LIN {X 0,Y 298.545,Z 280.112,A -85,B 0,C 180,E1 -16213.618,E2 -16213.618} C_VEL
LIN {X 0,Y 298.541,Z 280.111,A -85,B 0,C 180,E1 -16216.411,E2 -16216.411} C_VEL
LIN {X 0,Y 298.503,Z 280.117,A -85,B 0,C 180,E1 -16219.656,E2 -16219.656} C_VEL
LIN {X 0,Y 298.417,Z 280.126,A -85,B 0,C 180,E1 -16223.603,E2 -16223.603} C_VEL
LIN {X 0,Y 298.403,Z 280.131,A -85,B 0,C 180,E1 -16226.585,E2 -16226.585} C_VEL
LIN {X 0,Y 298.388,Z 280.134,A -85,B 0,C 180,E1 -16229.647,E2 -16229.647} C_VEL
LIN {X 0,Y 298.388,Z 280.135,A -85,B 0,C 180,E1 -16232.803,E2 -16232.803} C_VEL
LIN {X 0,Y 298.461,Z 280.124,A -85,B 0,C 180,E1 -16236.815,E2 -16236.815} C_VEL
LIN {X 0,Y 298.415,Z 280.127,A -85,B 0,C 180,E1 -16241.097,E2 -16241.097} C_VEL
LIN {X 0,Y 298.427,Z 280.25,A -85,B 0,C 180,E1 -16243.54,E2 -16243.54} C_VEL
LIN {X 0,Y 299.046,Z 283.99,A -85,B 0,C 180,E1 -16247.039,E2 -16247.039} C_VEL
LIN {X 0,Y 299.67,Z 287.19,A -85,B 0,C 180,E1 -16249.842,E2 -16249.842} C_VEL
LIN {X 0,Y 300.261,Z 290.689,A -85,B 0,C 180,E1 -16252.735,E2 -16252.735} C_VEL
LIN {X 0,Y 300.627,Z 293.494,A -85,B 0,C 180,E1 -16254.91,E2 -16254.91} C_VEL
LIN {X 0,Y 300.519,Z 296.811,A -85,B 0,C 180,E1 -16257.344,E2 -16257.344} C_VEL
LIN {X 0,Y 299.5,Z 302.518,A -85,B 0,C 180,E1 -16261.248,E2 -16261.248} C_VEL
LIN {X 0,Y 298.415,Z 309.186,A -85,B 0,C 180,E1 -16265.663,E2 -16265.663} C_VEL
LIN {X 0,Y 297.791,Z 313.823,A -85,B 0,C 180,E1 -16268.636,E2 -16268.636} C_VEL
LIN {X 0,Y 300.523,Z 326.073,A -85,B 0,C 180,E1 -16269.564,E2 -16269.564} C_VEL
LIN {X 0,Y 302.121,Z 336.168,A -85,B 0,C 180,E1 -16270.52,E2 -16270.52} C_VEL
LIN {X 0,Y 302.918,Z 345.087,A -85,B 0,C 180,E1 -16271.519,E2 -16271.519} C_VEL
LIN {X 0,Y 303.106,Z 352.307,A -85,B 0,C 180,E1 -16272.459,E2 -16272.459} C_VEL
LIN {X 0,Y 302.625,Z 359.174,A -85,B 0,C 180,E1 -16273.474,E2 -16273.474} C_VEL
LIN {X 0,Y 301.244,Z 366.76,A -85,B 0,C 180,E1 -16274.786,E2 -16274.786} C_VEL
LIN {X 0,Y 300.07,Z 373.019,A -85,B 0,C 180,E1 -16276.111,E2 -16276.111} C_VEL
LIN {X 0,Y 299.132,Z 378.235,A -85,B 0,C 180,E1 -16277.45,E2 -16277.45} C_VEL
LIN {X 0,Y 298.133,Z 383.56,A -85,B 0,C 180,E1 -16279.132,E2 -16279.132} C_VEL
LIN {X 0,Y 297.531,Z 387.015,A -85,B 0,C 180,E1 -16280.484,E2 -16280.484} C_VEL
LIN {X 0,Y 296.906,Z 391.022,A -85,B 0,C 180,E1 -16282.521,E2 -16282.521} C_VEL
LIN {X 0,Y 296.605,Z 393.796,A -85,B 0,C 180,E1 -16284.563,E2 -16284.563} C_VEL
LIN {X 0,Y 296.606,Z 394.925,A -85,B 0,C 180,E1 -16285.926,E2 -16285.926} C_VEL
LIN {X 0,Y 296.591,Z 395.588,A -85,B 0,C 180,E1 -16287.285,E2 -16287.285} C_VEL
LIN {X 0,Y 296.599,Z 395.794,A -85,B 0,C 180,E1 -16288.644,E2 -16288.644} C_VEL
LIN {X 0,Y 296.676,Z 395.491,A -85,B 0,C 180,E1 -16290.002,E2 -16290.002} C_VEL
LIN {X 0,Y 296.641,Z 394.591,A -85,B 0,C 180,E1 -16291.359,E2 -16291.359} C_VEL
LIN {X 0,Y 296.633,Z 393.199,A -85,B 0,C 180,E1 -16292.718,E2 -16292.718} C_VEL
LIN {X 0,Y 296.668,Z 390.135,A -85,B 0,C 180,E1 -16294.758,E2 -16294.758} C_VEL
LIN {X 0,Y 296.805,Z 385.735,A -85,B 0,C 180,E1 -16296.801,E2 -16296.801} C_VEL
LIN {X 0,Y 297.112,Z 380.807,A -85,B 0,C 180,E1 -16298.503,E2 -16298.503} C_VEL
LIN {X 0,Y 297.524,Z 374.552,A -85,B 0,C 180,E1 -16300.206,E2 -16300.206} C_VEL
LIN {X 0,Y 298.089,Z 368.449,A -85,B 0,C 180,E1 -16301.562,E2 -16301.562} C_VEL
LIN {X 0,Y 298.72,Z 362.048,A -85,B 0,C 180,E1 -16302.744,E2 -16302.744} C_VEL
LIN {X 0,Y 299.405,Z 354.282,A -85,B 0,C 180,E1 -16303.924,E2 -16303.924} C_VEL
LIN {X 0,Y 299.61,Z 349.093,A -85,B 0,C 180,E1 -16304.607,E2 -16304.607} C_VEL
LIN {X 0,Y 299.163,Z 340.12,A -85,B 0,C 180,E1 -16305.592,E2 -16305.592} C_VEL
LIN {X 0,Y 298.532,Z 330.671,A -85,B 0,C 180,E1 -16306.411,E2 -16306.411} C_VEL
LIN {X 0,Y 297.725,Z 321.328,A -85,B 0,C 180,E1 -16307.031,E2 -16307.031} C_VEL
LIN {X 0,Y 296.991,Z 314.602,A -85,B 0,C 180,E1 -16307.385,E2 -16307.385} C_VEL
LIN {X 0,Y 297.477,Z 307.895,A -85,B 0,C 180,E1 -16311.483,E2 -16311.483} C_VEL
LIN {X 0,Y 298.201,Z 300.922,A -85,B 0,C 180,E1 -16315.785,E2 -16315.785} C_VEL
LIN {X 0,Y 299.154,Z 293.722,A -85,B 0,C 180,E1 -16320.34,E2 -16320.34} C_VEL
LIN {X 0,Y 299.771,Z 290.127,A -85,B 0,C 180,E1 -16322.633,E2 -16322.633} C_VEL
LIN {X 0,Y 299.704,Z 286.87,A -85,B 0,C 180,E1 -16324.838,E2 -16324.838} C_VEL
LIN {X 0,Y 298.969,Z 282.858,A -85,B 0,C 180,E1 -16327.678,E2 -16327.678} C_VEL
LIN {X 0,Y 298.502,Z 280.116,A -85,B 0,C 180,E1 -16329.692,E2 -16329.692} C_VEL
LIN {X 0,Y 298.41,Z 280.124,A -85,B 0,C 180,E1 -16333.103,E2 -16333.103} C_VEL
LIN {X 0,Y 298.414,Z 280.123,A -85,B 0,C 180,E1 -16336.921,E2 -16336.921} C_VEL
LIN {X 0,Y 298.415,Z 280.123,A -85,B 0,C 180,E1 -16341.006,E2 -16341.006} C_VEL
LIN {X 0,Y 298.429,Z 280.124,A -85,B 0,C 180,E1 -16343.93,E2 -16343.93} C_VEL
LIN {X 0,Y 298.406,Z 280.125,A -85,B 0,C 180,E1 -16347.983,E2 -16347.983} C_VEL
LIN {X 0,Y 298.474,Z 280.117,A -85,B 0,C 180,E1 -16351.903,E2 -16351.903} C_VEL
LIN {X 0,Y 298.494,Z 280.115,A -85,B 0,C 180,E1 -16354.923,E2 -16354.923} C_VEL
LIN {X 0,Y 298.433,Z 280.125,A -85,B 0,C 180,E1 -16359.312,E2 -16359.312} C_VEL
LIN {X 0,Y 298.476,Z 280.115,A -85,B 0,C 180,E1 -16362.173,E2 -16362.173} C_VEL
LIN {X 0,Y 298.595,Z 280.105,A -85,B 0,C 180,E1 -16364.993,E2 -16364.993} C_VEL
LIN {X 0,Y 298.592,Z 280.103,A -85,B 0,C 180,E1 -16369.144,E2 -16369.144} C_VEL
LIN {X 0,Y 298.726,Z 280.084,A -85,B 0,C 180,E1 -16371.883,E2 -16371.883} C_VEL
LIN {X 0,Y 298.66,Z 280.096,A -85,B 0,C 180,E1 -16374.597,E2 -16374.597} C_VEL
LIN {X 0,Y 298.929,Z 280.062,A -85,B 0,C 180,E1 -16378.65,E2 -16378.65} C_VEL
LIN {X 0,Y 298.93,Z 280.058,A -85,B 0,C 180,E1 -16381.345,E2 -16381.345} C_VEL
LIN {X 0,Y 298.803,Z 280.076,A -85,B 0,C 180,E1 -16386.751,E2 -16386.751} C_VEL
LIN {X 0,Y 298.685,Z 280.088,A -85,B 0,C 180,E1 -16389.478,E2 -16389.478} C_VEL
LIN {X 0,Y 298.555,Z 280.106,A -85,B 0,C 180,E1 -16393.612,E2 -16393.612} C_VEL
LIN {X 0,Y 298.551,Z 280.109,A -85,B 0,C 180,E1 -16396.406,E2 -16396.406} C_VEL
LIN {X 0,Y 298.513,Z 280.112,A -85,B 0,C 180,E1 -16399.651,E2 -16399.651} C_VEL
LIN {X 0,Y 298.458,Z 280.119,A -85,B 0,C 180,E1 -16403.594,E2 -16403.594} C_VEL
LIN {X 0,Y 298.486,Z 280.114,A -85,B 0,C 180,E1 -16406.571,E2 -16406.571} C_VEL
LIN {X 0,Y 298.414,Z 280.127,A -85,B 0,C 180,E1 -16409.638,E2 -16409.638} C_VEL
LIN {X 0,Y 298.392,Z 280.126,A -85,B 0,C 180,E1 -16412.797,E2 -16412.797} C_VEL
LIN {X 0,Y 298.467,Z 280.117,A -85,B 0,C 180,E1 -16416.81,E2 -16416.81} C_VEL
LIN {X 0,Y 298.451,Z 280.122,A -85,B 0,C 180,E1 -16421.246,E2 -16421.246} C_VEL
LIN {X 0,Y 298.483,Z 280.118,A -85,B 0,C 180,E1 -16425.057,E2 -16425.057} C_VEL
LIN {X 0,Y 298.445,Z 280.122,A -85,B 0,C 180,E1 -16428.895,E2 -16428.895} C_VEL
LIN {X 0,Y 298.456,Z 280.121,A -85,B 0,C 180,E1 -16433.184,E2 -16433.184} C_VEL
LIN {X 0,Y 298.385,Z 280.129,A -85,B 0,C 180,E1 -16437.197,E2 -16437.197} C_VEL
LIN {X 0,Y 298.42,Z 280.126,A -85,B 0,C 180,E1 -16440.612,E2 -16440.612} C_VEL
LIN {X 0,Y 298.472,Z 280.116,A -85,B 0,C 180,E1 -16443.471,E2 -16443.471} C_VEL
LIN {X 0,Y 298.425,Z 280.126,A -85,B 0,C 180,E1 -16446.693,E2 -16446.693} C_VEL
LIN {X 0,Y 298.418,Z 280.125,A -85,B 0,C 180,E1 -16450.747,E2 -16450.747} C_VEL
LIN {X 0,Y 298.015,Z 280.174,A -85,B 0,C 180,E1 -16454.963,E2 -16454.963} C_VEL
LIN {X 0,Y 297.655,Z 280.391,A -85,B 0,C 180,E1 -16457.383,E2 -16457.383} C_VEL
LIN {X 0,Y 297.631,Z 285.417,A -85,B 0,C 180,E1 -16462.607,E2 -16462.607} C_VEL
LIN {X 0,Y 297.388,Z 289.552,A -85,B 0,C 180,E1 -16466.781,E2 -16466.781} C_VEL
LIN {X 0,Y 299.242,Z 300.537,A -85,B 0,C 180,E1 -16467.474,E2 -16467.474} C_VEL
LIN {X 0,Y 300.308,Z 308.84,A -85,B 0,C 180,E1 -16468.154,E2 -16468.154} C_VEL
LIN {X 0,Y 301.049,Z 315.665,A -85,B 0,C 180,E1 -16468.828,E2 -16468.828} C_VEL
LIN {X 0,Y 300.195,Z 325.606,A -85,B 0,C 180,E1 -16469.998,E2 -16469.998} C_VEL
LIN {X 0,Y 299.521,Z 333.548,A -85,B 0,C 180,E1 -16471.175,E2 -16471.175} C_VEL
LIN {X 0,Y 298.889,Z 340.115,A -85,B 0,C 180,E1 -16472.357,E2 -16472.357} C_VEL
LIN {X 0,Y 298.325,Z 346.345,A -85,B 0,C 180,E1 -16473.713,E2 -16473.713} C_VEL
LIN {X 0,Y 297.802,Z 351.531,A -85,B 0,C 180,E1 -16475.075,E2 -16475.075} C_VEL
LIN {X 0,Y 297.633,Z 354.859,A -85,B 0,C 180,E1 -16476.098,E2 -16476.098} C_VEL
LIN {X 0,Y 297.239,Z 358.487,A -85,B 0,C 180,E1 -16477.402,E2 -16477.402} C_VEL
LIN {X 0,Y 296.95,Z 361.721,A -85,B 0,C 180,E1 -16478.847,E2 -16478.847} C_VEL
LIN {X 0,Y 296.613,Z 365.121,A -85,B 0,C 180,E1 -16480.925,E2 -16480.925} C_VEL
LIN {X 0,Y 296.56,Z 366.746,A -85,B 0,C 180,E1 -16482.313,E2 -16482.313} C_VEL
LIN {X 0,Y 296.574,Z 367.763,A -85,B 0,C 180,E1 -16483.706,E2 -16483.706} C_VEL
LIN {X 0,Y 296.595,Z 368.251,A -85,B 0,C 180,E1 -16485.107,E2 -16485.107} C_VEL
LIN {X 0,Y 296.691,Z 368.247,A -85,B 0,C 180,E1 -16486.512,E2 -16486.512} C_VEL
LIN {X 0,Y 297.176,Z 367.049,A -85,B 0,C 180,E1 -16488.931,E2 -16488.931} C_VEL
LIN {X 0,Y 297.711,Z 365.089,A -85,B 0,C 180,E1 -16490.736,E2 -16490.736} C_VEL
LIN {X 0,Y 298.515,Z 361.625,A -85,B 0,C 180,E1 -16492.807,E2 -16492.807} C_VEL
LIN {X 0,Y 299.211,Z 358.347,A -85,B 0,C 180,E1 -16494.268,E2 -16494.268} C_VEL
LIN {X 0,Y 300.29,Z 353.239,A -85,B 0,C 180,E1 -16496.027,E2 -16496.027} C_VEL
LIN {X 0,Y 301.416,Z 347.367,A -85,B 0,C 180,E1 -16497.629,E2 -16497.629} C_VEL
LIN {X 0,Y 302.411,Z 342.037,A -85,B 0,C 180,E1 -16498.829,E2 -16498.829} C_VEL
LIN {X 0,Y 303.72,Z 334.476,A -85,B 0,C 180,E1 -16500.216,E2 -16500.216} C_VEL
LIN {X 0,Y 304.891,Z 327.594,A -85,B 0,C 180,E1 -16501.243,E2 -16501.243} C_VEL
LIN {X 0,Y 305.508,Z 322.294,A -85,B 0,C 180,E1 -16501.942,E2 -16501.942} C_VEL
LIN {X 0,Y 304.004,Z 313.232,A -85,B 0,C 180,E1 -16503.109,E2 -16503.109} C_VEL
LIN {X 0,Y 302.018,Z 304.972,A -85,B 0,C 180,E1 -16504.039,E2 -16504.039} C_VEL
LIN {X 0,Y 299.205,Z 295.676,A -85,B 0,C 180,E1 -16504.94,E2 -16504.94} C_VEL
LIN {X 0,Y 297.573,Z 290.412,A -85,B 0,C 180,E1 -16505.398,E2 -16505.398} C_VEL
LIN {X 0,Y 297.897,Z 286.701,A -85,B 0,C 180,E1 -16509.565,E2 -16509.565} C_VEL
LIN {X 0,Y 298.214,Z 283.678,A -85,B 0,C 180,E1 -16513.11,E2 -16513.11} C_VEL
LIN {X 0,Y 298.281,Z 282.127,A -85,B 0,C 180,E1 -16515.026,E2 -16515.026} C_VEL
LIN {X 0,Y 298.269,Z 280.606,A -85,B 0,C 180,E1 -16516.92,E2 -16516.92} C_VEL
LIN {X 0,Y 298.312,Z 280.14,A -85,B 0,C 180,E1 -16518.926,E2 -16518.926} C_VEL
LIN {X 0,Y 298.412,Z 280.13,A -85,B 0,C 180,E1 -16522.246,E2 -16522.246} C_VEL
LIN {X 0,Y 298.39,Z 280.131,A -85,B 0,C 180,E1 -16525.582,E2 -16525.582} C_VEL
LIN {X 0,Y 298.374,Z 280.132,A -85,B 0,C 180,E1 -16528.792,E2 -16528.792} C_VEL
LIN {X 0,Y 298.441,Z 280.123,A -85,B 0,C 180,E1 -16531.905,E2 -16531.905} C_VEL
LIN {X 0,Y 298.467,Z 280.12,A -85,B 0,C 180,E1 -16534.926,E2 -16534.926} C_VEL
LIN {X 0,Y 298.425,Z 280.121,A -85,B 0,C 180,E1 -16539.317,E2 -16539.317} C_VEL
LIN {X 0,Y 298.522,Z 280.108,A -85,B 0,C 180,E1 -16542.181,E2 -16542.181} C_VEL
LIN {X 0,Y 298.579,Z 280.103,A -85,B 0,C 180,E1 -16544.997,E2 -16544.997} C_VEL
LIN {X 0,Y 298.58,Z 280.102,A -85,B 0,C 180,E1 -16549.149,E2 -16549.149} C_VEL
LIN {X 0,Y 298.699,Z 280.09,A -85,B 0,C 180,E1 -16551.887,E2 -16551.887} C_VEL
LIN {X 0,Y 298.619,Z 280.097,A -85,B 0,C 180,E1 -16554.756,E2 -16554.756} C_VEL
LIN {X 0,Y 297.938,Z 280.187,A -85,B 0,C 180,E1 -16555.884,E2 -16555.884} C_VEL
LIN {X 0,Y 295.241,Z 280.518,A -85,B 0,C 180,E1 -16557.727,E2 -16557.727} C_VEL
LIN {X 0,Y 292.973,Z 280.803,A -85,B 0,C 180,E1 -16559.221,E2 -16559.221} C_VEL
LIN {X 0,Y 291.984,Z 280.928,A -85,B 0,C 180,E1 -16560.374,E2 -16560.374} C_VEL
LIN {X 0,Y 291.892,Z 280.934,A -85,B 0,C 180,E1 -16560.764,E2 -16560.764} C_VEL
LIN {X 0,Y 291.778,Z 280.95,A -85,B 0,C 180,E1 -16562.764,E2 -16562.764} C_VEL
LIN {X 0,Y 291.737,Z 280.954,A -85,B 0,C 180,E1 -16566.92,E2 -16566.92} C_VEL
LIN {X 0,Y 291.621,Z 280.972,A -85,B 0,C 180,E1 -16569.714,E2 -16569.714} C_VEL
LIN {X 0,Y 291.515,Z 280.986,A -85,B 0,C 180,E1 -16573.953,E2 -16573.953} C_VEL
LIN {X 0,Y 291.479,Z 280.99,A -85,B 0,C 180,E1 -16576.821,E2 -16576.821} C_VEL
LIN {X 0,Y 291.444,Z 280.995,A -85,B 0,C 180,E1 -16579.878,E2 -16579.878} C_VEL
LIN {X 0,Y 291.358,Z 281.007,A -85,B 0,C 180,E1 -16584.211,E2 -16584.211} C_VEL
LIN {X 0,Y 291.348,Z 281.01,A -85,B 0,C 180,E1 -16587.281,E2 -16587.281} C_VEL
LIN {X 0,Y 291.313,Z 281.016,A -85,B 0,C 180,E1 -16590.442,E2 -16590.442} C_VEL
LIN {X 0,Y 291.339,Z 281.014,A -85,B 0,C 180,E1 -16593.701,E2 -16593.701} C_VEL
LIN {X 0,Y 291.394,Z 281.005,A -85,B 0,C 180,E1 -16597.262,E2 -16597.262} C_VEL
LIN {X 0,Y 291.373,Z 281.004,A -85,B 0,C 180,E1 -16600.638,E2 -16600.638} C_VEL
LIN {X 0,Y 291.378,Z 281.017,A -85,B 0,C 180,E1 -16602.787,E2 -16602.787} C_VEL
LIN {X 0,Y 291.913,Z 284.561,A -85,B 0,C 180,E1 -16606.245,E2 -16606.245} C_VEL
LIN {X 0,Y 292.766,Z 288.957,A -85,B 0,C 180,E1 -16610.193,E2 -16610.193} C_VEL
LIN {X 0,Y 293.361,Z 292.55,A -85,B 0,C 180,E1 -16613.21,E2 -16613.21} C_VEL
LIN {X 0,Y 293.643,Z 295.809,A -85,B 0,C 180,E1 -16615.777,E2 -16615.777} C_VEL
LIN {X 0,Y 293.591,Z 297.336,A -85,B 0,C 180,E1 -16616.915,E2 -16616.915} C_VEL
LIN {X 0,Y 292.643,Z 302.424,A -85,B 0,C 180,E1 -16620.518,E2 -16620.518} C_VEL
LIN {X 0,Y 291.66,Z 307.954,A -85,B 0,C 180,E1 -16624.297,E2 -16624.297} C_VEL
LIN {X 0,Y 290.867,Z 313.615,A -85,B 0,C 180,E1 -16627.985,E2 -16627.985} C_VEL
LIN {X 0,Y 293.687,Z 326.04,A -85,B 0,C 180,E1 -16628.966,E2 -16628.966} C_VEL
LIN {X 0,Y 295.19,Z 335.075,A -85,B 0,C 180,E1 -16629.847,E2 -16629.847} C_VEL
LIN {X 0,Y 296.117,Z 344.757,A -85,B 0,C 180,E1 -16630.962,E2 -16630.962} C_VEL
LIN {X 0,Y 296.39,Z 351.078,A -85,B 0,C 180,E1 -16631.801,E2 -16631.801} C_VEL
LIN {X 0,Y 295.995,Z 358.469,A -85,B 0,C 180,E1 -16632.915,E2 -16632.915} C_VEL
LIN {X 0,Y 294.773,Z 365.263,A -85,B 0,C 180,E1 -16634.089,E2 -16634.089} C_VEL
LIN {X 0,Y 293.462,Z 371.716,A -85,B 0,C 180,E1 -16635.438,E2 -16635.438} C_VEL
LIN {X 0,Y 292.411,Z 377.098,A -85,B 0,C 180,E1 -16636.803,E2 -16636.803} C_VEL
LIN {X 0,Y 291.538,Z 381.61,A -85,B 0,C 180,E1 -16638.178,E2 -16638.178} C_VEL
LIN {X 0,Y 290.806,Z 385.383,A -85,B 0,C 180,E1 -16639.559,E2 -16639.559} C_VEL
LIN {X 0,Y 290.037,Z 389.701,A -85,B 0,C 180,E1 -16641.642,E2 -16641.642} C_VEL
LIN {X 0,Y 289.723,Z 391.935,A -85,B 0,C 180,E1 -16643.035,E2 -16643.035} C_VEL
LIN {X 0,Y 289.522,Z 393.585,A -85,B 0,C 180,E1 -16644.43,E2 -16644.43} C_VEL
LIN {X 0,Y 289.503,Z 394.666,A -85,B 0,C 180,E1 -16645.825,E2 -16645.825} C_VEL
LIN {X 0,Y 289.517,Z 395.282,A -85,B 0,C 180,E1 -16647.219,E2 -16647.219} C_VEL
LIN {X 0,Y 289.515,Z 395.439,A -85,B 0,C 180,E1 -16648.611,E2 -16648.611} C_VEL
LIN {X 0,Y 289.586,Z 395.117,A -85,B 0,C 180,E1 -16650.002,E2 -16650.002} C_VEL
LIN {X 0,Y 289.555,Z 394.189,A -85,B 0,C 180,E1 -16651.393,E2 -16651.393} C_VEL
LIN {X 0,Y 289.561,Z 392.748,A -85,B 0,C 180,E1 -16652.784,E2 -16652.784} C_VEL
LIN {X 0,Y 289.554,Z 389.152,A -85,B 0,C 180,E1 -16655.152,E2 -16655.152} C_VEL
LIN {X 0,Y 289.745,Z 385.137,A -85,B 0,C 180,E1 -16656.968,E2 -16656.968} C_VEL
LIN {X 0,Y 290.083,Z 380.125,A -85,B 0,C 180,E1 -16658.711,E2 -16658.711} C_VEL
LIN {X 0,Y 290.524,Z 373.796,A -85,B 0,C 180,E1 -16660.455,E2 -16660.455} C_VEL
LIN {X 0,Y 291.092,Z 367.602,A -85,B 0,C 180,E1 -16661.844,E2 -16661.844} C_VEL
LIN {X 0,Y 291.74,Z 361.093,A -85,B 0,C 180,E1 -16663.054,E2 -16663.054} C_VEL
LIN {X 0,Y 292.501,Z 353.204,A -85,B 0,C 180,E1 -16664.259,E2 -16664.259} C_VEL
LIN {X 0,Y 292.503,Z 347.805,A -85,B 0,C 180,E1 -16664.97,E2 -16664.97} C_VEL
LIN {X 0,Y 292.021,Z 338.601,A -85,B 0,C 180,E1 -16665.98,E2 -16665.98} C_VEL
LIN {X 0,Y 291.457,Z 329.842,A -85,B 0,C 180,E1 -16666.742,E2 -16666.742} C_VEL
LIN {X 0,Y 290.599,Z 320.471,A -85,B 0,C 180,E1 -16667.371,E2 -16667.371} C_VEL
LIN {X 0,Y 289.935,Z 314.237,A -85,B 0,C 180,E1 -16667.731,E2 -16667.731} C_VEL
LIN {X 0,Y 290.484,Z 307.412,A -85,B 0,C 180,E1 -16672.027,E2 -16672.027} C_VEL
LIN {X 0,Y 291.128,Z 301.549,A -85,B 0,C 180,E1 -16675.757,E2 -16675.757} C_VEL
LIN {X 0,Y 292.101,Z 294.449,A -85,B 0,C 180,E1 -16680.351,E2 -16680.351} C_VEL
LIN {X 0,Y 292.73,Z 290.693,A -85,B 0,C 180,E1 -16682.826,E2 -16682.826} C_VEL
LIN {X 0,Y 292.571,Z 287.238,A -85,B 0,C 180,E1 -16685.239,E2 -16685.239} C_VEL
LIN {X 0,Y 291.512,Z 281.433,A -85,B 0,C 180,E1 -16689.51,E2 -16689.51} C_VEL
LIN {X 0,Y 291.422,Z 280.999,A -85,B 0,C 180,E1 -16690.011,E2 -16690.011} C_VEL
LIN {X 0,Y 291.301,Z 281.011,A -85,B 0,C 180,E1 -16694.402,E2 -16694.402} C_VEL
LIN {X 0,Y 291.337,Z 281.006,A -85,B 0,C 180,E1 -16698.404,E2 -16698.404} C_VEL
LIN {X 0,Y 291.364,Z 281.002,A -85,B 0,C 180,E1 -16701.158,E2 -16701.158} C_VEL
LIN {X 0,Y 291.372,Z 281,A -85,B 0,C 180,E1 -16704.625,E2 -16704.625} C_VEL
LIN {X 0,Y 291.383,Z 281,A -85,B 0,C 180,E1 -16707.95,E2 -16707.95} C_VEL
LIN {X 0,Y 291.393,Z 280.999,A -85,B 0,C 180,E1 -16711.157,E2 -16711.157} C_VEL
LIN {X 0,Y 291.426,Z 280.993,A -85,B 0,C 180,E1 -16714.271,E2 -16714.271} C_VEL
LIN {X 0,Y 291.382,Z 281.002,A -85,B 0,C 180,E1 -16717.297,E2 -16717.297} C_VEL
LIN {X 0,Y 291.416,Z 280.994,A -85,B 0,C 180,E1 -16720.265,E2 -16720.265} C_VEL
LIN {X 0,Y 291.507,Z 280.985,A -85,B 0,C 180,E1 -16724.664,E2 -16724.664} C_VEL
LIN {X 0,Y 291.538,Z 280.982,A -85,B 0,C 180,E1 -16728.878,E2 -16728.878} C_VEL
LIN {X 0,Y 291.676,Z 280.962,A -85,B 0,C 180,E1 -16731.685,E2 -16731.685} C_VEL
LIN {X 0,Y 291.63,Z 280.971,A -85,B 0,C 180,E1 -16734.466,E2 -16734.466} C_VEL
LIN {X 0,Y 291.895,Z 280.938,A -85,B 0,C 180,E1 -16738.618,E2 -16738.618} C_VEL
LIN {X 0,Y 291.897,Z 280.934,A -85,B 0,C 180,E1 -16741.377,E2 -16741.377} C_VEL
LIN {X 0,Y 291.752,Z 280.954,A -85,B 0,C 180,E1 -16746.915,E2 -16746.915} C_VEL
LIN {X 0,Y 291.634,Z 280.967,A -85,B 0,C 180,E1 -16749.709,E2 -16749.709} C_VEL
LIN {X 0,Y 291.525,Z 280.983,A -85,B 0,C 180,E1 -16753.947,E2 -16753.947} C_VEL
LIN {X 0,Y 291.49,Z 280.986,A -85,B 0,C 180,E1 -16756.815,E2 -16756.815} C_VEL
LIN {X 0,Y 291.453,Z 280.993,A -85,B 0,C 180,E1 -16759.872,E2 -16759.872} C_VEL
LIN {X 0,Y 291.401,Z 280.999,A -85,B 0,C 180,E1 -16764.202,E2 -16764.202} C_VEL
LIN {X 0,Y 291.419,Z 280.996,A -85,B 0,C 180,E1 -16767.268,E2 -16767.268} C_VEL
LIN {X 0,Y 291.332,Z 281.005,A -85,B 0,C 180,E1 -16770.434,E2 -16770.434} C_VEL
LIN {X 0,Y 291.342,Z 281.008,A -85,B 0,C 180,E1 -16773.695,E2 -16773.695} C_VEL
LIN {X 0,Y 291.401,Z 280.999,A -85,B 0,C 180,E1 -16777.258,E2 -16777.258} C_VEL
LIN {X 0,Y 291.401,Z 280.996,A -85,B 0,C 180,E1 -16780.627,E2 -16780.627} C_VEL
LIN {X 0,Y 291.4,Z 280.997,A -85,B 0,C 180,E1 -16784.376,E2 -16784.376} C_VEL
LIN {X 0,Y 291.381,Z 280.999,A -85,B 0,C 180,E1 -16788.387,E2 -16788.387} C_VEL
LIN {X 0,Y 291.371,Z 281.005,A -85,B 0,C 180,E1 -16791.159,E2 -16791.159} C_VEL
LIN {X 0,Y 291.375,Z 281.002,A -85,B 0,C 180,E1 -16794.626,E2 -16794.626} C_VEL
LIN {X 0,Y 291.361,Z 281.001,A -85,B 0,C 180,E1 -16797.948,E2 -16797.948} C_VEL
LIN {X 0,Y 291.371,Z 281.002,A -85,B 0,C 180,E1 -16801.155,E2 -16801.155} C_VEL
LIN {X 0,Y 291.405,Z 280.998,A -85,B 0,C 180,E1 -16804.269,E2 -16804.269} C_VEL
LIN {X 0,Y 291.367,Z 281.001,A -85,B 0,C 180,E1 -16807.297,E2 -16807.297} C_VEL
LIN {X 0,Y 291.369,Z 281.004,A -85,B 0,C 180,E1 -16810.262,E2 -16810.262} C_VEL
LIN {X 0,Y 290.993,Z 281.051,A -85,B 0,C 180,E1 -16814.592,E2 -16814.592} C_VEL
LIN {X 0,Y 290.585,Z 281.213,A -85,B 0,C 180,E1 -16817.426,E2 -16817.426} C_VEL
LIN {X 0,Y 290.563,Z 286.088,A -85,B 0,C 180,E1 -16822.579,E2 -16822.579} C_VEL
LIN {X 0,Y 290.369,Z 289.861,A -85,B 0,C 180,E1 -16826.442,E2 -16826.442} C_VEL
LIN {X 0,Y 292.323,Z 301.667,A -85,B 0,C 180,E1 -16827.242,E2 -16827.242} C_VEL
LIN {X 0,Y 293.359,Z 309.794,A -85,B 0,C 180,E1 -16827.939,E2 -16827.939} C_VEL
LIN {X 0,Y 294.047,Z 316.52,A -85,B 0,C 180,E1 -16828.629,E2 -16828.629} C_VEL
LIN {X 0,Y 293.321,Z 325.118,A -85,B 0,C 180,E1 -16829.655,E2 -16829.655} C_VEL
LIN {X 0,Y 292.595,Z 333.205,A -85,B 0,C 180,E1 -16830.858,E2 -16830.858} C_VEL
LIN {X 0,Y 291.92,Z 339.886,A -85,B 0,C 180,E1 -16832.068,E2 -16832.068} C_VEL
LIN {X 0,Y 291.326,Z 346.211,A -85,B 0,C 180,E1 -16833.456,E2 -16833.456} C_VEL
LIN {X 0,Y 290.769,Z 351.478,A -85,B 0,C 180,E1 -16834.851,E2 -16834.851} C_VEL
LIN {X 0,Y 290.487,Z 355.845,A -85,B 0,C 180,E1 -16836.248,E2 -16836.248} C_VEL
LIN {X 0,Y 289.953,Z 361.042,A -85,B 0,C 180,E1 -16838.36,E2 -16838.36} C_VEL
LIN {X 0,Y 289.59,Z 364.845,A -85,B 0,C 180,E1 -16840.485,E2 -16840.485} C_VEL
LIN {X 0,Y 289.457,Z 367.262,A -85,B 0,C 180,E1 -16842.62,E2 -16842.62} C_VEL
LIN {X 0,Y 289.494,Z 368.25,A -85,B 0,C 180,E1 -16844.048,E2 -16844.048} C_VEL
LIN {X 0,Y 289.525,Z 368.644,A -85,B 0,C 180,E1 -16845.485,E2 -16845.485} C_VEL
LIN {X 0,Y 289.653,Z 368.529,A -85,B 0,C 180,E1 -16846.925,E2 -16846.925} C_VEL
LIN {X 0,Y 290.155,Z 367.379,A -85,B 0,C 180,E1 -16849.165,E2 -16849.165} C_VEL
LIN {X 0,Y 290.797,Z 365.109,A -85,B 0,C 180,E1 -16851.253,E2 -16851.253} C_VEL
LIN {X 0,Y 291.634,Z 361.712,A -85,B 0,C 180,E1 -16853.241,E2 -16853.241} C_VEL
LIN {X 0,Y 292.478,Z 358.029,A -85,B 0,C 180,E1 -16854.865,E2 -16854.865} C_VEL
LIN {X 0,Y 293.622,Z 352.755,A -85,B 0,C 180,E1 -16856.664,E2 -16856.664} C_VEL
LIN {X 0,Y 294.653,Z 347.692,A -85,B 0,C 180,E1 -16858.06,E2 -16858.06} C_VEL
LIN {X 0,Y 295.932,Z 341.181,A -85,B 0,C 180,E1 -16859.521,E2 -16859.521} C_VEL
LIN {X 0,Y 297.149,Z 334.443,A -85,B 0,C 180,E1 -16860.759,E2 -16860.759} C_VEL
LIN {X 0,Y 298.437,Z 327.036,A -85,B 0,C 180,E1 -16861.869,E2 -16861.869} C_VEL
LIN {X 0,Y 298.829,Z 324.368,A -85,B 0,C 180,E1 -16862.236,E2 -16862.236} C_VEL
LIN {X 0,Y 297.319,Z 314.591,A -85,B 0,C 180,E1 -16863.57,E2 -16863.57} C_VEL
LIN {X 0,Y 295.405,Z 306.371,A -85,B 0,C 180,E1 -16864.543,E2 -16864.543} C_VEL
LIN {X 0,Y 292.317,Z 296.166,A -85,B 0,C 180,E1 -16865.581,E2 -16865.581} C_VEL
LIN {X 0,Y 290.588,Z 290.763,A -85,B 0,C 180,E1 -16866.071,E2 -16866.071} C_VEL
LIN {X 0,Y 290.847,Z 287.887,A -85,B 0,C 180,E1 -16869.359,E2 -16869.359} C_VEL
LIN {X 0,Y 291.11,Z 285.246,A -85,B 0,C 180,E1 -16872.527,E2 -16872.527} C_VEL
LIN {X 0,Y 291.237,Z 282.787,A -85,B 0,C 180,E1 -16875.593,E2 -16875.593} C_VEL
LIN {X 0,Y 291.211,Z 281.315,A -85,B 0,C 180,E1 -16877.492,E2 -16877.492} C_VEL
LIN {X 0,Y 291.273,Z 281.018,A -85,B 0,C 180,E1 -16879.352,E2 -16879.352} C_VEL
LIN {X 0,Y 291.406,Z 281.003,A -85,B 0,C 180,E1 -16882.923,E2 -16882.923} C_VEL
LIN {X 0,Y 291.326,Z 281.011,A -85,B 0,C 180,E1 -16886.303,E2 -16886.303} C_VEL
LIN {X 0,Y 291.366,Z 281.005,A -85,B 0,C 180,E1 -16890.263,E2 -16890.263} C_VEL
LIN {X 0,Y 291.397,Z 281.001,A -85,B 0,C 180,E1 -16894.273,E2 -16894.273} C_VEL
LIN {X 0,Y 291.359,Z 281.006,A -85,B 0,C 180,E1 -16897.301,E2 -16897.301} C_VEL
LIN {X 0,Y 291.443,Z 280.996,A -85,B 0,C 180,E1 -16900.272,E2 -16900.272} C_VEL
LIN {X 0,Y 291.541,Z 280.983,A -85,B 0,C 180,E1 -16904.626,E2 -16904.626} C_VEL
LIN {X 0,Y 291.524,Z 280.982,A -85,B 0,C 180,E1 -16908.883,E2 -16908.883} C_VEL
LIN {X 0,Y 291.65,Z 280.969,A -85,B 0,C 180,E1 -16911.689,E2 -16911.689} C_VEL
LIN {X 0,Y 291.576,Z 280.973,A -85,B 0,C 180,E1 -16914.734,E2 -16914.734} C_VEL
LIN {X 0,Y 291.88,Z 280.935,A -85,B 0,C 180,E1 -16918.623,E2 -16918.623} C_VEL
LIN {X 0,Y 291.892,Z 280.934,A -85,B 0,C 180,E1 -16920.764,E2 -16920.764} C_VEL
LIN {X 0,Y 291.155,Z 281.027,A -85,B 0,C 180,E1 -16921.913,E2 -16921.913} C_VEL
LIN {X 0,Y 288.163,Z 281.404,A -85,B 0,C 180,E1 -16923.78,E2 -16923.78} C_VEL
LIN {X 0,Y 285.695,Z 281.707,A -85,B 0,C 180,E1 -16925.296,E2 -16925.296} C_VEL
LIN {X 0,Y 284.706,Z 281.827,A -85,B 0,C 180,E1 -16926.473,E2 -16926.473} C_VEL
LIN {X 0,Y 284.663,Z 281.834,A -85,B 0,C 180,E1 -16926.872,E2 -16926.872} C_VEL
LIN {X 0,Y 284.558,Z 281.853,A -85,B 0,C 180,E1 -16929.958,E2 -16929.958} C_VEL
LIN {X 0,Y 284.474,Z 281.863,A -85,B 0,C 180,E1 -16934.305,E2 -16934.305} C_VEL
LIN {X 0,Y 284.418,Z 281.869,A -85,B 0,C 180,E1 -16937.251,E2 -16937.251} C_VEL
LIN {X 0,Y 284.371,Z 281.875,A -85,B 0,C 180,E1 -16940.245,E2 -16940.245} C_VEL
LIN {X 0,Y 284.318,Z 281.883,A -85,B 0,C 180,E1 -16943.857,E2 -16943.857} C_VEL
LIN {X 0,Y 284.278,Z 281.891,A -85,B 0,C 180,E1 -16948.019,E2 -16948.019} C_VEL
LIN {X 0,Y 284.28,Z 281.892,A -85,B 0,C 180,E1 -16951.278,E2 -16951.278} C_VEL
LIN {X 0,Y 284.358,Z 281.882,A -85,B 0,C 180,E1 -16955.357,E2 -16955.357} C_VEL
LIN {X 0,Y 284.326,Z 281.884,A -85,B 0,C 180,E1 -16958.169,E2 -16958.169} C_VEL
LIN {X 0,Y 284.305,Z 281.885,A -85,B 0,C 180,E1 -16962.076,E2 -16962.076} C_VEL
LIN {X 0,Y 284.868,Z 285.418,A -85,B 0,C 180,E1 -16965.683,E2 -16965.683} C_VEL
LIN {X 0,Y 285.696,Z 289.696,A -85,B 0,C 180,E1 -16969.695,E2 -16969.695} C_VEL
LIN {X 0,Y 286.342,Z 293.583,A -85,B 0,C 180,E1 -16973.038,E2 -16973.038} C_VEL
LIN {X 0,Y 286.642,Z 296.829,A -85,B 0,C 180,E1 -16975.675,E2 -16975.675} C_VEL
LIN {X 0,Y 286.434,Z 299.034,A -85,B 0,C 180,E1 -16977.333,E2 -16977.333} C_VEL
LIN {X 0,Y 285.392,Z 304.536,A -85,B 0,C 180,E1 -16981.304,E2 -16981.304} C_VEL
LIN {X 0,Y 284.379,Z 310.052,A -85,B 0,C 180,E1 -16985.159,E2 -16985.159} C_VEL
LIN {X 0,Y 283.911,Z 313.158,A -85,B 0,C 180,E1 -16987.272,E2 -16987.272} C_VEL
LIN {X 0,Y 286.647,Z 325.055,A -85,B 0,C 180,E1 -16988.235,E2 -16988.235} C_VEL
LIN {X 0,Y 288.253,Z 334.09,A -85,B 0,C 180,E1 -16989.143,E2 -16989.143} C_VEL
LIN {X 0,Y 289.298,Z 343.967,A -85,B 0,C 180,E1 -16990.315,E2 -16990.315} C_VEL
LIN {X 0,Y 289.616,Z 351.763,A -85,B 0,C 180,E1 -16991.396,E2 -16991.396} C_VEL
LIN {X 0,Y 289.221,Z 358.78,A -85,B 0,C 180,E1 -16992.502,E2 -16992.502} C_VEL
LIN {X 0,Y 287.957,Z 365.468,A -85,B 0,C 180,E1 -16993.702,E2 -16993.702} C_VEL
LIN {X 0,Y 286.586,Z 371.831,A -85,B 0,C 180,E1 -16995.081,E2 -16995.081} C_VEL
LIN {X 0,Y 285.504,Z 377.136,A -85,B 0,C 180,E1 -16996.478,E2 -16996.478} C_VEL
LIN {X 0,Y 284.572,Z 381.579,A -85,B 0,C 180,E1 -16997.884,E2 -16997.884} C_VEL
LIN {X 0,Y 283.492,Z 386.826,A -85,B 0,C 180,E1 -17000.009,E2 -17000.009} C_VEL
LIN {X 0,Y 282.994,Z 389.55,A -85,B 0,C 180,E1 -17001.433,E2 -17001.433} C_VEL
LIN {X 0,Y 282.672,Z 391.73,A -85,B 0,C 180,E1 -17002.861,E2 -17002.861} C_VEL
LIN {X 0,Y 282.423,Z 393.558,A -85,B 0,C 180,E1 -17004.508,E2 -17004.508} C_VEL
LIN {X 0,Y 282.405,Z 394.41,A -85,B 0,C 180,E1 -17005.72,E2 -17005.72} C_VEL
LIN {X 0,Y 282.443,Z 394.976,A -85,B 0,C 180,E1 -17007.149,E2 -17007.149} C_VEL
LIN {X 0,Y 282.433,Z 395.083,A -85,B 0,C 180,E1 -17008.576,E2 -17008.576} C_VEL
LIN {X 0,Y 282.499,Z 394.727,A -85,B 0,C 180,E1 -17010.002,E2 -17010.002} C_VEL
LIN {X 0,Y 282.472,Z 393.783,A -85,B 0,C 180,E1 -17011.428,E2 -17011.428} C_VEL
LIN {X 0,Y 282.49,Z 391.428,A -85,B 0,C 180,E1 -17013.568,E2 -17013.568} C_VEL
LIN {X 0,Y 282.497,Z 387.701,A -85,B 0,C 180,E1 -17015.713,E2 -17015.713} C_VEL
LIN {X 0,Y 282.686,Z 384.507,A -85,B 0,C 180,E1 -17017.143,E2 -17017.143} C_VEL
LIN {X 0,Y 283.035,Z 379.42,A -85,B 0,C 180,E1 -17018.93,E2 -17018.93} C_VEL
LIN {X 0,Y 283.37,Z 374.442,A -85,B 0,C 180,E1 -17020.361,E2 -17020.361} C_VEL
LIN {X 0,Y 283.956,Z 368.447,A -85,B 0,C 180,E1 -17021.784,E2 -17021.784} C_VEL
LIN {X 0,Y 284.691,Z 361.141,A -85,B 0,C 180,E1 -17023.202,E2 -17023.202} C_VEL
LIN {X 0,Y 285.464,Z 353.328,A -85,B 0,C 180,E1 -17024.436,E2 -17024.436} C_VEL
LIN {X 0,Y 285.39,Z 346.476,A -85,B 0,C 180,E1 -17025.353,E2 -17025.353} C_VEL
LIN {X 0,Y 284.978,Z 338.499,A -85,B 0,C 180,E1 -17026.246,E2 -17026.246} C_VEL
LIN {X 0,Y 284.396,Z 329.298,A -85,B 0,C 180,E1 -17027.067,E2 -17027.067} C_VEL
LIN {X 0,Y 283.506,Z 319.622,A -85,B 0,C 180,E1 -17027.727,E2 -17027.727} C_VEL
LIN {X 0,Y 282.863,Z 313.979,A -85,B 0,C 180,E1 -17028.049,E2 -17028.049} C_VEL
LIN {X 0,Y 283.484,Z 306.941,A -85,B 0,C 180,E1 -17032.6,E2 -17032.6} C_VEL
LIN {X 0,Y 284.29,Z 300.013,A -85,B 0,C 180,E1 -17037.128,E2 -17037.128} C_VEL
LIN {X 0,Y 285.437,Z 292.807,A -85,B 0,C 180,E1 -17041.965,E2 -17041.965} C_VEL
LIN {X 0,Y 285.713,Z 290.959,A -85,B 0,C 180,E1 -17043.242,E2 -17043.242} C_VEL
LIN {X 0,Y 285.306,Z 286.804,A -85,B 0,C 180,E1 -17046.244,E2 -17046.244} C_VEL
LIN {X 0,Y 284.385,Z 281.875,A -85,B 0,C 180,E1 -17050.087,E2 -17050.087} C_VEL
LIN {X 0,Y 284.257,Z 281.889,A -85,B 0,C 180,E1 -17054.19,E2 -17054.19} C_VEL
LIN {X 0,Y 284.283,Z 281.886,A -85,B 0,C 180,E1 -17058.124,E2 -17058.124} C_VEL
LIN {X 0,Y 284.333,Z 281.877,A -85,B 0,C 180,E1 -17062.278,E2 -17062.278} C_VEL
LIN {X 0,Y 284.32,Z 281.881,A -85,B 0,C 180,E1 -17065.35,E2 -17065.35} C_VEL
LIN {X 0,Y 284.307,Z 281.879,A -85,B 0,C 180,E1 -17068.725,E2 -17068.725} C_VEL
LIN {X 0,Y 284.408,Z 281.868,A -85,B 0,C 180,E1 -17072.825,E2 -17072.825} C_VEL
LIN {X 0,Y 284.343,Z 281.875,A -85,B 0,C 180,E1 -17076.703,E2 -17076.703} C_VEL
LIN {X 0,Y 284.386,Z 281.87,A -85,B 0,C 180,E1 -17079.903,E2 -17079.903} C_VEL
LIN {X 0,Y 284.456,Z 281.863,A -85,B 0,C 180,E1 -17084.491,E2 -17084.491} C_VEL
LIN {X 0,Y 284.475,Z 281.859,A -85,B 0,C 180,E1 -17088.599,E2 -17088.599} C_VEL
LIN {X 0,Y 284.63,Z 281.841,A -85,B 0,C 180,E1 -17091.478,E2 -17091.478} C_VEL
LIN {X 0,Y 284.6,Z 281.845,A -85,B 0,C 180,E1 -17094.329,E2 -17094.329} C_VEL
LIN {X 0,Y 284.861,Z 281.813,A -85,B 0,C 180,E1 -17098.584,E2 -17098.584} C_VEL
LIN {X 0,Y 284.863,Z 281.81,A -85,B 0,C 180,E1 -17101.411,E2 -17101.411} C_VEL
LIN {X 0,Y 284.704,Z 281.831,A -85,B 0,C 180,E1 -17107.087,E2 -17107.087} C_VEL
LIN {X 0,Y 284.571,Z 281.847,A -85,B 0,C 180,E1 -17109.952,E2 -17109.952} C_VEL
LIN {X 0,Y 284.482,Z 281.863,A -85,B 0,C 180,E1 -17114.3,E2 -17114.3} C_VEL
LIN {X 0,Y 284.428,Z 281.865,A -85,B 0,C 180,E1 -17117.245,E2 -17117.245} C_VEL
LIN {X 0,Y 284.381,Z 281.872,A -85,B 0,C 180,E1 -17120.239,E2 -17120.239} C_VEL
LIN {X 0,Y 284.37,Z 281.875,A -85,B 0,C 180,E1 -17123.872,E2 -17123.872} C_VEL
LIN {X 0,Y 284.395,Z 281.87,A -85,B 0,C 180,E1 -17127.169,E2 -17127.169} C_VEL
LIN {X 0,Y 284.291,Z 281.884,A -85,B 0,C 180,E1 -17131.271,E2 -17131.271} C_VEL
LIN {X 0,Y 284.359,Z 281.877,A -85,B 0,C 180,E1 -17135.351,E2 -17135.351} C_VEL
LIN {X 0,Y 284.334,Z 281.878,A -85,B 0,C 180,E1 -17138.161,E2 -17138.161} C_VEL
LIN {X 0,Y 284.339,Z 281.877,A -85,B 0,C 180,E1 -17142.138,E2 -17142.138} C_VEL
LIN {X 0,Y 284.346,Z 281.875,A -85,B 0,C 180,E1 -17146.205,E2 -17146.205} C_VEL
LIN {X 0,Y 284.343,Z 281.875,A -85,B 0,C 180,E1 -17150.01,E2 -17150.01} C_VEL
LIN {X 0,Y 284.343,Z 281.876,A -85,B 0,C 180,E1 -17153.614,E2 -17153.614} C_VEL
LIN {X 0,Y 284.297,Z 281.884,A -85,B 0,C 180,E1 -17157.186,E2 -17157.186} C_VEL
LIN {X 0,Y 284.347,Z 281.877,A -85,B 0,C 180,E1 -17160.373,E2 -17160.373} C_VEL
LIN {X 0,Y 284.366,Z 281.873,A -85,B 0,C 180,E1 -17163.584,E2 -17163.584} C_VEL
LIN {X 0,Y 284.354,Z 281.879,A -85,B 0,C 180,E1 -17166.704,E2 -17166.704} C_VEL
LIN {X 0,Y 284.32,Z 281.88,A -85,B 0,C 180,E1 -17169.925,E2 -17169.925} C_VEL
LIN {X 0,Y 283.986,Z 281.924,A -85,B 0,C 180,E1 -17174.202,E2 -17174.202} C_VEL
LIN {X 0,Y 283.533,Z 282.04,A -85,B 0,C 180,E1 -17177.472,E2 -17177.472} C_VEL
LIN {X 0,Y 283.512,Z 286.73,A -85,B 0,C 180,E1 -17182.523,E2 -17182.523} C_VEL
LIN {X 0,Y 283.337,Z 290.2,A -85,B 0,C 180,E1 -17186.131,E2 -17186.131} C_VEL
LIN {X 0,Y 285.229,Z 301.714,A -85,B 0,C 180,E1 -17186.908,E2 -17186.908} C_VEL
LIN {X 0,Y 286.395,Z 310.755,A -85,B 0,C 180,E1 -17187.713,E2 -17187.713} C_VEL
LIN {X 0,Y 287.087,Z 315.857,A -85,B 0,C 180,E1 -17188.245,E2 -17188.245} C_VEL
LIN {X 0,Y 286.313,Z 325.866,A -85,B 0,C 180,E1 -17189.471,E2 -17189.471} C_VEL
LIN {X 0,Y 285.637,Z 332.863,A -85,B 0,C 180,E1 -17190.527,E2 -17190.527} C_VEL
LIN {X 0,Y 284.958,Z 339.65,A -85,B 0,C 180,E1 -17191.765,E2 -17191.765} C_VEL
LIN {X 0,Y 284.324,Z 346.07,A -85,B 0,C 180,E1 -17193.186,E2 -17193.186} C_VEL
LIN {X 0,Y 283.764,Z 351.414,A -85,B 0,C 180,E1 -17194.615,E2 -17194.615} C_VEL
LIN {X 0,Y 283.374,Z 356.587,A -85,B 0,C 180,E1 -17196.318,E2 -17196.318} C_VEL
LIN {X 0,Y 282.971,Z 360.345,A -85,B 0,C 180,E1 -17197.849,E2 -17197.849} C_VEL
LIN {X 0,Y 282.567,Z 364.398,A -85,B 0,C 180,E1 -17200.025,E2 -17200.025} C_VEL
LIN {X 0,Y 282.406,Z 366.343,A -85,B 0,C 180,E1 -17201.482,E2 -17201.482} C_VEL
LIN {X 0,Y 282.4,Z 368.452,A -85,B 0,C 180,E1 -17203.948,E2 -17203.948} C_VEL
LIN {X 0,Y 282.463,Z 369.036,A -85,B 0,C 180,E1 -17205.882,E2 -17205.882} C_VEL
LIN {X 0,Y 282.637,Z 368.811,A -85,B 0,C 180,E1 -17207.359,E2 -17207.359} C_VEL
LIN {X 0,Y 283.119,Z 367.717,A -85,B 0,C 180,E1 -17209.399,E2 -17209.399} C_VEL
LIN {X 0,Y 283.916,Z 365.063,A -85,B 0,C 180,E1 -17211.794,E2 -17211.794} C_VEL
LIN {X 0,Y 284.572,Z 362.673,A -85,B 0,C 180,E1 -17213.273,E2 -17213.273} C_VEL
LIN {X 0,Y 285.757,Z 357.698,A -85,B 0,C 180,E1 -17215.491,E2 -17215.491} C_VEL
LIN {X 0,Y 286.729,Z 353.483,A -85,B 0,C 180,E1 -17216.963,E2 -17216.963} C_VEL
LIN {X 0,Y 287.892,Z 348.045,A -85,B 0,C 180,E1 -17218.506,E2 -17218.506} C_VEL
LIN {X 0,Y 289.148,Z 342.096,A -85,B 0,C 180,E1 -17219.883,E2 -17219.883} C_VEL
LIN {X 0,Y 290.406,Z 335.478,A -85,B 0,C 180,E1 -17221.148,E2 -17221.148} C_VEL
LIN {X 0,Y 291.806,Z 327.82,A -85,B 0,C 180,E1 -17222.337,E2 -17222.337} C_VEL
LIN {X 0,Y 292.137,Z 325.57,A -85,B 0,C 180,E1 -17222.654,E2 -17222.654} C_VEL
LIN {X 0,Y 290.973,Z 317.41,A -85,B 0,C 180,E1 -17223.849,E2 -17223.849} C_VEL
LIN {X 0,Y 288.775,Z 307.656,A -85,B 0,C 180,E1 -17225.087,E2 -17225.087} C_VEL
LIN {X 0,Y 285.445,Z 296.764,A -85,B 0,C 180,E1 -17226.248,E2 -17226.248} C_VEL
LIN {X 0,Y 283.598,Z 291.096,A -85,B 0,C 180,E1 -17226.787,E2 -17226.787} C_VEL
LIN {X 0,Y 283.852,Z 288.327,A -85,B 0,C 180,E1 -17230.069,E2 -17230.069} C_VEL
LIN {X 0,Y 284.173,Z 285.297,A -85,B 0,C 180,E1 -17233.824,E2 -17233.824} C_VEL
LIN {X 0,Y 284.234,Z 283.443,A -85,B 0,C 180,E1 -17236.19,E2 -17236.19} C_VEL
LIN {X 0,Y 284.178,Z 282.016,A -85,B 0,C 180,E1 -17238.112,E2 -17238.112} C_VEL
LIN {X 0,Y 284.285,Z 281.887,A -85,B 0,C 180,E1 -17240.026,E2 -17240.026} C_VEL
LIN {X 0,Y 284.332,Z 281.884,A -85,B 0,C 180,E1 -17243.618,E2 -17243.618} C_VEL
LIN {X 0,Y 284.289,Z 281.886,A -85,B 0,C 180,E1 -17247.191,E2 -17247.191} C_VEL
LIN {X 0,Y 284.338,Z 281.882,A -85,B 0,C 180,E1 -17250.377,E2 -17250.377} C_VEL
LIN {X 0,Y 284.359,Z 281.876,A -85,B 0,C 180,E1 -17253.588,E2 -17253.588} C_VEL
LIN {X 0,Y 284.317,Z 281.88,A -85,B 0,C 180,E1 -17256.706,E2 -17256.706} C_VEL
LIN {X 0,Y 284.388,Z 281.874,A -85,B 0,C 180,E1 -17261.264,E2 -17261.264} C_VEL
LIN {X 0,Y 284.478,Z 281.863,A -85,B 0,C 180,E1 -17264.461,E2 -17264.461} C_VEL
LIN {X 0,Y 284.476,Z 281.86,A -85,B 0,C 180,E1 -17268.604,E2 -17268.604} C_VEL
LIN {X 0,Y 284.606,Z 281.847,A -85,B 0,C 180,E1 -17271.482,E2 -17271.482} C_VEL
LIN {X 0,Y 284.57,Z 281.845,A -85,B 0,C 180,E1 -17274.333,E2 -17274.333} C_VEL
LIN {X 0,Y 284.846,Z 281.811,A -85,B 0,C 180,E1 -17278.589,E2 -17278.589} C_VEL
LIN {X 0,Y 284.845,Z 281.812,A -85,B 0,C 180,E1 -17281.416,E2 -17281.416} C_VEL
LIN {X 0,Y 284.663,Z 281.834,A -85,B 0,C 180,E1 -17286.872,E2 -17286.872} C_VEL
LIN {X 0,Y 284.056,Z 281.916,A -85,B 0,C 180,E1 -17288.051,E2 -17288.051} C_VEL
LIN {X 0,Y 281.096,Z 282.284,A -85,B 0,C 180,E1 -17289.968,E2 -17289.968} C_VEL
LIN {X 0,Y 278.546,Z 282.601,A -85,B 0,C 180,E1 -17291.526,E2 -17291.526} C_VEL
LIN {X 0,Y 277.477,Z 282.734,A -85,B 0,C 180,E1 -17292.737,E2 -17292.737} C_VEL
LIN {X 0,Y 277.408,Z 282.743,A -85,B 0,C 180,E1 -17293.148,E2 -17293.148} C_VEL
LIN {X 0,Y 277.399,Z 282.745,A -85,B 0,C 180,E1 -17296.184,E2 -17296.184} C_VEL
LIN {X 0,Y 277.338,Z 282.751,A -85,B 0,C 180,E1 -17300.352,E2 -17300.352} C_VEL
LIN {X 0,Y 277.274,Z 282.761,A -85,B 0,C 180,E1 -17304.155,E2 -17304.155} C_VEL
LIN {X 0,Y 277.265,Z 282.766,A -85,B 0,C 180,E1 -17307.486,E2 -17307.486} C_VEL
LIN {X 0,Y 277.243,Z 282.77,A -85,B 0,C 180,E1 -17310.476,E2 -17310.476} C_VEL
LIN {X 0,Y 277.25,Z 282.769,A -85,B 0,C 180,E1 -17313.898,E2 -17313.898} C_VEL
LIN {X 0,Y 277.282,Z 282.762,A -85,B 0,C 180,E1 -17317.469,E2 -17317.469} C_VEL
LIN {X 0,Y 277.294,Z 282.952,A -85,B 0,C 180,E1 -17321.605,E2 -17321.605} C_VEL
LIN {X 0,Y 277.829,Z 286.259,A -85,B 0,C 180,E1 -17325.099,E2 -17325.099} C_VEL
LIN {X 0,Y 278.604,Z 290.504,A -85,B 0,C 180,E1 -17329.183,E2 -17329.183} C_VEL
LIN {X 0,Y 279.327,Z 294.593,A -85,B 0,C 180,E1 -17332.857,E2 -17332.857} C_VEL
LIN {X 0,Y 279.602,Z 296.764,A -85,B 0,C 180,E1 -17334.684,E2 -17334.684} C_VEL
LIN {X 0,Y 279.631,Z 298.942,A -85,B 0,C 180,E1 -17336.434,E2 -17336.434} C_VEL
LIN {X 0,Y 278.739,Z 303.318,A -85,B 0,C 180,E1 -17339.719,E2 -17339.719} C_VEL
LIN {X 0,Y 277.66,Z 308.811,A -85,B 0,C 180,E1 -17343.71,E2 -17343.71} C_VEL
LIN {X 0,Y 276.996,Z 312.788,A -85,B 0,C 180,E1 -17346.523,E2 -17346.523} C_VEL
LIN {X 0,Y 278.968,Z 321.096,A -85,B 0,C 180,E1 -17347.205,E2 -17347.205} C_VEL
LIN {X 0,Y 281.252,Z 332.512,A -85,B 0,C 180,E1 -17348.333,E2 -17348.333} C_VEL
LIN {X 0,Y 282.458,Z 343.094,A -85,B 0,C 180,E1 -17349.616,E2 -17349.616} C_VEL
LIN {X 0,Y 282.813,Z 351.37,A -85,B 0,C 180,E1 -17350.793,E2 -17350.793} C_VEL
LIN {X 0,Y 282.584,Z 358.107,A -85,B 0,C 180,E1 -17351.89,E2 -17351.89} C_VEL
LIN {X 0,Y 281.621,Z 363.989,A -85,B 0,C 180,E1 -17352.951,E2 -17352.951} C_VEL
LIN {X 0,Y 280.074,Z 370.541,A -85,B 0,C 180,E1 -17354.352,E2 -17354.352} C_VEL
LIN {X 0,Y 278.831,Z 376.007,A -85,B 0,C 180,E1 -17355.776,E2 -17355.776} C_VEL
LIN {X 0,Y 277.628,Z 381.551,A -85,B 0,C 180,E1 -17357.576,E2 -17357.576} C_VEL
LIN {X 0,Y 276.493,Z 386.734,A -85,B 0,C 180,E1 -17359.753,E2 -17359.753} C_VEL
LIN {X 0,Y 275.756,Z 390.567,A -85,B 0,C 180,E1 -17361.944,E2 -17361.944} C_VEL
LIN {X 0,Y 275.346,Z 393.426,A -85,B 0,C 180,E1 -17364.545,E2 -17364.545} C_VEL
LIN {X 0,Y 275.311,Z 394.154,A -85,B 0,C 180,E1 -17365.61,E2 -17365.61} C_VEL
LIN {X 0,Y 275.369,Z 394.671,A -85,B 0,C 180,E1 -17367.076,E2 -17367.076} C_VEL
LIN {X 0,Y 275.354,Z 394.727,A -85,B 0,C 180,E1 -17368.539,E2 -17368.539} C_VEL
LIN {X 0,Y 275.414,Z 394.326,A -85,B 0,C 180,E1 -17370.002,E2 -17370.002} C_VEL
LIN {X 0,Y 275.392,Z 393.374,A -85,B 0,C 180,E1 -17371.464,E2 -17371.464} C_VEL
LIN {X 0,Y 275.411,Z 390.924,A -85,B 0,C 180,E1 -17373.66,E2 -17373.66} C_VEL
LIN {X 0,Y 275.425,Z 387.129,A -85,B 0,C 180,E1 -17375.86,E2 -17375.86} C_VEL
LIN {X 0,Y 275.763,Z 381.941,A -85,B 0,C 180,E1 -17378.06,E2 -17378.06} C_VEL
LIN {X 0,Y 276.159,Z 376.341,A -85,B 0,C 180,E1 -17379.893,E2 -17379.893} C_VEL
LIN {X 0,Y 276.828,Z 369.287,A -85,B 0,C 180,E1 -17381.72,E2 -17381.72} C_VEL
LIN {X 0,Y 277.644,Z 361.189,A -85,B 0,C 180,E1 -17383.357,E2 -17383.357} C_VEL
LIN {X 0,Y 278.439,Z 353.453,A -85,B 0,C 180,E1 -17384.622,E2 -17384.622} C_VEL
LIN {X 0,Y 278.345,Z 346.716,A -85,B 0,C 180,E1 -17385.561,E2 -17385.561} C_VEL
LIN {X 0,Y 277.94,Z 337.686,A -85,B 0,C 180,E1 -17386.595,E2 -17386.595} C_VEL
LIN {X 0,Y 277.316,Z 328.595,A -85,B 0,C 180,E1 -17387.421,E2 -17387.421} C_VEL
LIN {X 0,Y 276.409,Z 318.756,A -85,B 0,C 180,E1 -17388.102,E2 -17388.102} C_VEL
LIN {X 0,Y 275.828,Z 313.68,A -85,B 0,C 180,E1 -17388.381,E2 -17388.381} C_VEL
LIN {X 0,Y 276.471,Z 306.562,A -85,B 0,C 180,E1 -17393.128,E2 -17393.128} C_VEL
LIN {X 0,Y 277.287,Z 300.107,A -85,B 0,C 180,E1 -17397.486,E2 -17397.486} C_VEL
LIN {X 0,Y 278.388,Z 293.552,A -85,B 0,C 180,E1 -17402.018,E2 -17402.018} C_VEL
LIN {X 0,Y 278.648,Z 291.158,A -85,B 0,C 180,E1 -17403.704,E2 -17403.704} C_VEL
LIN {X 0,Y 278.323,Z 287.951,A -85,B 0,C 180,E1 -17406.092,E2 -17406.092} C_VEL
LIN {X 0,Y 277.359,Z 282.751,A -85,B 0,C 180,E1 -17410.209,E2 -17410.209} C_VEL
LIN {X 0,Y 277.212,Z 282.764,A -85,B 0,C 180,E1 -17414.773,E2 -17414.773} C_VEL
LIN {X 0,Y 277.221,Z 282.763,A -85,B 0,C 180,E1 -17418.763,E2 -17418.763} C_VEL
LIN {X 0,Y 277.278,Z 282.755,A -85,B 0,C 180,E1 -17422.53,E2 -17422.53} C_VEL
LIN {X 0,Y 277.258,Z 282.76,A -85,B 0,C 180,E1 -17426.104,E2 -17426.104} C_VEL
LIN {X 0,Y 277.273,Z 282.759,A -85,B 0,C 180,E1 -17429.538,E2 -17429.538} C_VEL
LIN {X 0,Y 277.37,Z 282.745,A -85,B 0,C 180,E1 -17432.863,E2 -17432.863} C_VEL
LIN {X 0,Y 277.308,Z 282.751,A -85,B 0,C 180,E1 -17436.075,E2 -17436.075} C_VEL
LIN {X 0,Y 277.315,Z 282.752,A -85,B 0,C 180,E1 -17440.762,E2 -17440.762} C_VEL
LIN {X 0,Y 277.419,Z 282.74,A -85,B 0,C 180,E1 -17445.323,E2 -17445.323} C_VEL
LIN {X 0,Y 277.464,Z 282.732,A -85,B 0,C 180,E1 -17449.785,E2 -17449.785} C_VEL
LIN {X 0,Y 277.636,Z 282.715,A -85,B 0,C 180,E1 -17452.726,E2 -17452.726} C_VEL
LIN {X 0,Y 277.827,Z 282.689,A -85,B 0,C 180,E1 -17458.548,E2 -17458.548} C_VEL
LIN {X 0,Y 277.829,Z 282.686,A -85,B 0,C 180,E1 -17461.447,E2 -17461.447} C_VEL
LIN {X 0,Y 277.659,Z 282.708,A -85,B 0,C 180,E1 -17467.268,E2 -17467.268} C_VEL
LIN {X 0,Y 277.512,Z 282.728,A -85,B 0,C 180,E1 -17470.208,E2 -17470.208} C_VEL
LIN {X 0,Y 277.432,Z 282.738,A -85,B 0,C 180,E1 -17474.671,E2 -17474.671} C_VEL
LIN {X 0,Y 277.347,Z 282.747,A -85,B 0,C 180,E1 -17479.23,E2 -17479.23} C_VEL
LIN {X 0,Y 277.32,Z 282.753,A -85,B 0,C 180,E1 -17484.167,E2 -17484.167} C_VEL
LIN {X 0,Y 277.323,Z 282.753,A -85,B 0,C 180,E1 -17487.501,E2 -17487.501} C_VEL
LIN {X 0,Y 277.271,Z 282.757,A -85,B 0,C 180,E1 -17490.478,E2 -17490.478} C_VEL
LIN {X 0,Y 277.251,Z 282.761,A -85,B 0,C 180,E1 -17493.891,E2 -17493.891} C_VEL
LIN {X 0,Y 277.288,Z 282.759,A -85,B 0,C 180,E1 -17497.462,E2 -17497.462} C_VEL
LIN {X 0,Y 277.289,Z 282.757,A -85,B 0,C 180,E1 -17501.218,E2 -17501.218} C_VEL
LIN {X 0,Y 277.282,Z 282.76,A -85,B 0,C 180,E1 -17505.205,E2 -17505.205} C_VEL
LIN {X 0,Y 277.287,Z 282.756,A -85,B 0,C 180,E1 -17509.491,E2 -17509.491} C_VEL
LIN {X 0,Y 277.277,Z 282.757,A -85,B 0,C 180,E1 -17512.53,E2 -17512.53} C_VEL
LIN {X 0,Y 277.244,Z 282.76,A -85,B 0,C 180,E1 -17516.102,E2 -17516.102} C_VEL
LIN {X 0,Y 277.251,Z 282.76,A -85,B 0,C 180,E1 -17519.535,E2 -17519.535} C_VEL
LIN {X 0,Y 277.347,Z 282.751,A -85,B 0,C 180,E1 -17522.861,E2 -17522.861} C_VEL
LIN {X 0,Y 277.317,Z 282.752,A -85,B 0,C 180,E1 -17526.077,E2 -17526.077} C_VEL
LIN {X 0,Y 277.261,Z 282.759,A -85,B 0,C 180,E1 -17529.687,E2 -17529.687} C_VEL
LIN {X 0,Y 276.969,Z 282.796,A -85,B 0,C 180,E1 -17533.79,E2 -17533.79} C_VEL
LIN {X 0,Y 276.539,Z 282.852,A -85,B 0,C 180,E1 -17537.15,E2 -17537.15} C_VEL
LIN {X 0,Y 276.472,Z 282.883,A -85,B 0,C 180,E1 -17537.52,E2 -17537.52} C_VEL
LIN {X 0,Y 276.446,Z 287.588,A -85,B 0,C 180,E1 -17542.695,E2 -17542.695} C_VEL
LIN {X 0,Y 276.29,Z 290.46,A -85,B 0,C 180,E1 -17545.759,E2 -17545.759} C_VEL
LIN {X 0,Y 278.336,Z 302.81,A -85,B 0,C 180,E1 -17546.651,E2 -17546.651} C_VEL
LIN {X 0,Y 279.443,Z 311.711,A -85,B 0,C 180,E1 -17547.476,E2 -17547.476} C_VEL
LIN {X 0,Y 280.113,Z 316.722,A -85,B 0,C 180,E1 -17548.021,E2 -17548.021} C_VEL
LIN {X 0,Y 279.303,Z 326.615,A -85,B 0,C 180,E1 -17549.277,E2 -17549.277} C_VEL
LIN {X 0,Y 278.609,Z 333.541,A -85,B 0,C 180,E1 -17550.359,E2 -17550.359} C_VEL
LIN {X 0,Y 278.022,Z 339.411,A -85,B 0,C 180,E1 -17551.447,E2 -17551.447} C_VEL
LIN {X 0,Y 277.329,Z 345.93,A -85,B 0,C 180,E1 -17552.903,E2 -17552.903} C_VEL
LIN {X 0,Y 276.749,Z 351.353,A -85,B 0,C 180,E1 -17554.367,E2 -17554.367} C_VEL
LIN {X 0,Y 276.428,Z 355.863,A -85,B 0,C 180,E1 -17555.835,E2 -17555.835} C_VEL
LIN {X 0,Y 275.995,Z 359.649,A -85,B 0,C 180,E1 -17557.313,E2 -17557.313} C_VEL
LIN {X 0,Y 275.705,Z 362.723,A -85,B 0,C 180,E1 -17558.796,E2 -17558.796} C_VEL
LIN {X 0,Y 275.439,Z 365.125,A -85,B 0,C 180,E1 -17560.287,E2 -17560.287} C_VEL
LIN {X 0,Y 275.292,Z 366.955,A -85,B 0,C 180,E1 -17561.783,E2 -17561.783} C_VEL
LIN {X 0,Y 275.304,Z 368.79,A -85,B 0,C 180,E1 -17564.069,E2 -17564.069} C_VEL
LIN {X 0,Y 275.405,Z 369.385,A -85,B 0,C 180,E1 -17566.3,E2 -17566.3} C_VEL
LIN {X 0,Y 275.654,Z 369.093,A -85,B 0,C 180,E1 -17567.813,E2 -17567.813} C_VEL
LIN {X 0,Y 276.1,Z 368.052,A -85,B 0,C 180,E1 -17569.652,E2 -17569.652} C_VEL
LIN {X 0,Y 277.039,Z 365.003,A -85,B 0,C 180,E1 -17572.364,E2 -17572.364} C_VEL
LIN {X 0,Y 278.061,Z 361.199,A -85,B 0,C 180,E1 -17574.517,E2 -17574.517} C_VEL
LIN {X 0,Y 279.077,Z 357.38,A -85,B 0,C 180,E1 -17576.146,E2 -17576.146} C_VEL
LIN {X 0,Y 280.183,Z 353.021,A -85,B 0,C 180,E1 -17577.646,E2 -17577.646} C_VEL
LIN {X 0,Y 281.426,Z 347.199,A -85,B 0,C 180,E1 -17579.283,E2 -17579.283} C_VEL
LIN {X 0,Y 282.758,Z 341.272,A -85,B 0,C 180,E1 -17580.63,E2 -17580.63} C_VEL
LIN {X 0,Y 284.329,Z 333.37,A -85,B 0,C 180,E1 -17582.1,E2 -17582.1} C_VEL
LIN {X 0,Y 285.434,Z 326.352,A -85,B 0,C 180,E1 -17583.166,E2 -17583.166} C_VEL
LIN {X 0,Y 284.16,Z 318.064,A -85,B 0,C 180,E1 -17584.437,E2 -17584.437} C_VEL
LIN {X 0,Y 281.738,Z 307.419,A -85,B 0,C 180,E1 -17585.83,E2 -17585.83} C_VEL
LIN {X 0,Y 278.473,Z 297.039,A -85,B 0,C 180,E1 -17586.988,E2 -17586.988} C_VEL
LIN {X 0,Y 276.613,Z 291.444,A -85,B 0,C 180,E1 -17587.571,E2 -17587.571} C_VEL
LIN {X 0,Y 276.909,Z 288.386,A -85,B 0,C 180,E1 -17591.288,E2 -17591.288} C_VEL
LIN {X 0,Y 277.167,Z 285.651,A -85,B 0,C 180,E1 -17594.771,E2 -17594.771} C_VEL
LIN {X 0,Y 277.177,Z 283.752,A -85,B 0,C 180,E1 -17597.33,E2 -17597.33} C_VEL
LIN {X 0,Y 277.144,Z 282.777,A -85,B 0,C 180,E1 -17598.756,E2 -17598.756} C_VEL
LIN {X 0,Y 277.262,Z 282.766,A -85,B 0,C 180,E1 -17602.534,E2 -17602.534} C_VEL
LIN {X 0,Y 277.236,Z 282.765,A -85,B 0,C 180,E1 -17606.107,E2 -17606.107} C_VEL
LIN {X 0,Y 277.244,Z 282.763,A -85,B 0,C 180,E1 -17609.54,E2 -17609.54} C_VEL
LIN {X 0,Y 277.34,Z 282.751,A -85,B 0,C 180,E1 -17612.866,E2 -17612.866} C_VEL
LIN {X 0,Y 277.281,Z 282.755,A -85,B 0,C 180,E1 -17616.079,E2 -17616.079} C_VEL
LIN {X 0,Y 277.33,Z 282.753,A -85,B 0,C 180,E1 -17620.768,E2 -17620.768} C_VEL
LIN {X 0,Y 277.421,Z 282.736,A -85,B 0,C 180,E1 -17625.328,E2 -17625.328} C_VEL
LIN {X 0,Y 277.448,Z 282.732,A -85,B 0,C 180,E1 -17629.789,E2 -17629.789} C_VEL
LIN {X 0,Y 277.598,Z 282.716,A -85,B 0,C 180,E1 -17632.73,E2 -17632.73} C_VEL
LIN {X 0,Y 277.812,Z 282.687,A -85,B 0,C 180,E1 -17638.553,E2 -17638.553} C_VEL
LIN {X 0,Y 277.811,Z 282.688,A -85,B 0,C 180,E1 -17641.452,E2 -17641.452} C_VEL
LIN {X 0,Y 277.644,Z 282.712,A -85,B 0,C 180,E1 -17647.274,E2 -17647.274} C_VEL
LIN {X 0,Y 277.499,Z 282.734,A -85,B 0,C 180,E1 -17650.214,E2 -17650.214} C_VEL
LIN {X 0,Y 277.408,Z 282.743,A -85,B 0,C 180,E1 -17653.148,E2 -17653.148} C_VEL
LIN {X 0,Y 276.765,Z 282.828,A -85,B 0,C 180,E1 -17654.359,E2 -17654.359} C_VEL
LIN {X 0,Y 273.847,Z 283.188,A -85,B 0,C 180,E1 -17656.329,E2 -17656.329} C_VEL
LIN {X 0,Y 271.371,Z 283.496,A -85,B 0,C 180,E1 -17657.931,E2 -17657.931} C_VEL
LIN {X 0,Y 270.346,Z 283.622,A -85,B 0,C 180,E1 -17659.175,E2 -17659.175} C_VEL
LIN {X 0,Y 270.284,Z 283.63,A -85,B 0,C 180,E1 -17659.597,E2 -17659.597} C_VEL
LIN {X 0,Y 270.219,Z 283.643,A -85,B 0,C 180,E1 -17664.593,E2 -17664.593} C_VEL
LIN {X 0,Y 270.194,Z 283.647,A -85,B 0,C 180,E1 -17667.92,E2 -17667.92} C_VEL
LIN {X 0,Y 270.169,Z 283.65,A -85,B 0,C 180,E1 -17671.353,E2 -17671.353} C_VEL
LIN {X 0,Y 270.211,Z 283.646,A -85,B 0,C 180,E1 -17674.907,E2 -17674.907} C_VEL
LIN {X 0,Y 270.22,Z 283.64,A -85,B 0,C 180,E1 -17678.72,E2 -17678.72} C_VEL
LIN {X 0,Y 270.24,Z 283.714,A -85,B 0,C 180,E1 -17680.735,E2 -17680.735} C_VEL
LIN {X 0,Y 270.772,Z 287.113,A -85,B 0,C 180,E1 -17684.493,E2 -17684.493} C_VEL
LIN {X 0,Y 271.509,Z 291.284,A -85,B 0,C 180,E1 -17688.651,E2 -17688.651} C_VEL
LIN {X 0,Y 272.099,Z 294.536,A -85,B 0,C 180,E1 -17691.695,E2 -17691.695} C_VEL
LIN {X 0,Y 272.586,Z 297.788,A -85,B 0,C 180,E1 -17694.544,E2 -17694.544} C_VEL
LIN {X 0,Y 272.605,Z 300.047,A -85,B 0,C 180,E1 -17696.407,E2 -17696.407} C_VEL
LIN {X 0,Y 271.69,Z 304.308,A -85,B 0,C 180,E1 -17699.71,E2 -17699.71} C_VEL
LIN {X 0,Y 270.563,Z 309.795,A -85,B 0,C 180,E1 -17703.798,E2 -17703.798} C_VEL
LIN {X 0,Y 270.116,Z 312.584,A -85,B 0,C 180,E1 -17705.737,E2 -17705.737} C_VEL
LIN {X 0,Y 273.137,Z 325.455,A -85,B 0,C 180,E1 -17706.905,E2 -17706.905} C_VEL
LIN {X 0,Y 274.65,Z 333.696,A -85,B 0,C 180,E1 -17707.81,E2 -17707.81} C_VEL
LIN {X 0,Y 275.654,Z 342.301,A -85,B 0,C 180,E1 -17708.893,E2 -17708.893} C_VEL
LIN {X 0,Y 276.061,Z 350.829,A -85,B 0,C 180,E1 -17710.139,E2 -17710.139} C_VEL
LIN {X 0,Y 275.833,Z 358.485,A -85,B 0,C 180,E1 -17711.436,E2 -17711.436} C_VEL
LIN {X 0,Y 274.852,Z 364.223,A -85,B 0,C 180,E1 -17712.518,E2 -17712.518} C_VEL
LIN {X 0,Y 273.26,Z 370.68,A -85,B 0,C 180,E1 -17713.952,E2 -17713.952} C_VEL
LIN {X 0,Y 271.953,Z 376.065,A -85,B 0,C 180,E1 -17715.408,E2 -17715.408} C_VEL
LIN {X 0,Y 270.701,Z 381.537,A -85,B 0,C 180,E1 -17717.253,E2 -17717.253} C_VEL
LIN {X 0,Y 269.507,Z 386.653,A -85,B 0,C 180,E1 -17719.484,E2 -17719.484} C_VEL
LIN {X 0,Y 268.715,Z 390.422,A -85,B 0,C 180,E1 -17721.732,E2 -17721.732} C_VEL
LIN {X 0,Y 268.31,Z 392.896,A -85,B 0,C 180,E1 -17723.988,E2 -17723.988} C_VEL
LIN {X 0,Y 268.223,Z 393.899,A -85,B 0,C 180,E1 -17725.494,E2 -17725.494} C_VEL
LIN {X 0,Y 268.274,Z 394.365,A -85,B 0,C 180,E1 -17726.999,E2 -17726.999} C_VEL
LIN {X 0,Y 268.277,Z 394.372,A -85,B 0,C 180,E1 -17728.501,E2 -17728.501} C_VEL
LIN {X 0,Y 268.332,Z 393.919,A -85,B 0,C 180,E1 -17730.002,E2 -17730.002} C_VEL
LIN {X 0,Y 268.314,Z 392.953,A -85,B 0,C 180,E1 -17731.503,E2 -17731.503} C_VEL
LIN {X 0,Y 268.33,Z 390.411,A -85,B 0,C 180,E1 -17733.756,E2 -17733.756} C_VEL
LIN {X 0,Y 268.355,Z 386.557,A -85,B 0,C 180,E1 -17736.015,E2 -17736.015} C_VEL
LIN {X 0,Y 268.707,Z 381.305,A -85,B 0,C 180,E1 -17738.273,E2 -17738.273} C_VEL
LIN {X 0,Y 269.244,Z 374.309,A -85,B 0,C 180,E1 -17740.53,E2 -17740.53} C_VEL
LIN {X 0,Y 269.823,Z 368.412,A -85,B 0,C 180,E1 -17742.029,E2 -17742.029} C_VEL
LIN {X 0,Y 270.581,Z 361.227,A -85,B 0,C 180,E1 -17743.521,E2 -17743.521} C_VEL
LIN {X 0,Y 271.408,Z 353.567,A -85,B 0,C 180,E1 -17744.817,E2 -17744.817} C_VEL
LIN {X 0,Y 271.306,Z 346.365,A -85,B 0,C 180,E1 -17745.851,E2 -17745.851} C_VEL
LIN {X 0,Y 270.953,Z 338.673,A -85,B 0,C 180,E1 -17746.774,E2 -17746.774} C_VEL
LIN {X 0,Y 270.346,Z 329.08,A -85,B 0,C 180,E1 -17747.69,E2 -17747.69} C_VEL
LIN {X 0,Y 269.527,Z 319.981,A -85,B 0,C 180,E1 -17748.359,E2 -17748.359} C_VEL
LIN {X 0,Y 268.763,Z 313.329,A -85,B 0,C 180,E1 -17748.784,E2 -17748.784} C_VEL
LIN {X 0,Y 269.378,Z 307.123,A -85,B 0,C 180,E1 -17753.04,E2 -17753.04} C_VEL
LIN {X 0,Y 270.111,Z 301.339,A -85,B 0,C 180,E1 -17757.061,E2 -17757.061} C_VEL
LIN {X 0,Y 271.32,Z 294.257,A -85,B 0,C 180,E1 -17762.076,E2 -17762.076} C_VEL
LIN {X 0,Y 271.564,Z 291.488,A -85,B 0,C 180,E1 -17764.088,E2 -17764.088} C_VEL
LIN {X 0,Y 271.151,Z 288.265,A -85,B 0,C 180,E1 -17766.596,E2 -17766.596} C_VEL
LIN {X 0,Y 270.305,Z 283.628,A -85,B 0,C 180,E1 -17770.429,E2 -17770.429} C_VEL
LIN {X 0,Y 270.164,Z 283.643,A -85,B 0,C 180,E1 -17775.38,E2 -17775.38} C_VEL
LIN {X 0,Y 270.185,Z 283.642,A -85,B 0,C 180,E1 -17779.434,E2 -17779.434} C_VEL
LIN {X 0,Y 270.237,Z 283.637,A -85,B 0,C 180,E1 -17783.73,E2 -17783.73} C_VEL
LIN {X 0,Y 270.214,Z 283.636,A -85,B 0,C 180,E1 -17786.892,E2 -17786.892} C_VEL
LIN {X 0,Y 270.24,Z 283.631,A -85,B 0,C 180,E1 -17790.386,E2 -17790.386} C_VEL
LIN {X 0,Y 270.273,Z 283.63,A -85,B 0,C 180,E1 -17793.762,E2 -17793.762} C_VEL
LIN {X 0,Y 270.219,Z 283.636,A -85,B 0,C 180,E1 -17797.035,E2 -17797.035} C_VEL
LIN {X 0,Y 270.262,Z 283.629,A -85,B 0,C 180,E1 -17800.239,E2 -17800.239} C_VEL
LIN {X 0,Y 270.378,Z 283.619,A -85,B 0,C 180,E1 -17804.931,E2 -17804.931} C_VEL
LIN {X 0,Y 270.416,Z 283.61,A -85,B 0,C 180,E1 -17809.515,E2 -17809.515} C_VEL
LIN {X 0,Y 270.593,Z 283.591,A -85,B 0,C 180,E1 -17812.536,E2 -17812.536} C_VEL
LIN {X 0,Y 270.793,Z 283.565,A -85,B 0,C 180,E1 -17818.51,E2 -17818.51} C_VEL
LIN {X 0,Y 270.794,Z 283.563,A -85,B 0,C 180,E1 -17821.484,E2 -17821.484} C_VEL
LIN {X 0,Y 270.617,Z 283.585,A -85,B 0,C 180,E1 -17827.458,E2 -17827.458} C_VEL
LIN {X 0,Y 270.447,Z 283.607,A -85,B 0,C 180,E1 -17830.478,E2 -17830.478} C_VEL
LIN {X 0,Y 270.4,Z 283.613,A -85,B 0,C 180,E1 -17835.062,E2 -17835.062} C_VEL
LIN {X 0,Y 270.304,Z 283.626,A -85,B 0,C 180,E1 -17839.752,E2 -17839.752} C_VEL
LIN {X 0,Y 270.275,Z 283.628,A -85,B 0,C 180,E1 -17844.582,E2 -17844.582} C_VEL
LIN {X 0,Y 270.269,Z 283.633,A -85,B 0,C 180,E1 -17847.905,E2 -17847.905} C_VEL
LIN {X 0,Y 270.182,Z 283.642,A -85,B 0,C 180,E1 -17851.345,E2 -17851.345} C_VEL
LIN {X 0,Y 270.213,Z 283.636,A -85,B 0,C 180,E1 -17854.9,E2 -17854.9} C_VEL
LIN {X 0,Y 270.249,Z 283.632,A -85,B 0,C 180,E1 -17858.721,E2 -17858.721} C_VEL
LIN {X 0,Y 270.251,Z 283.632,A -85,B 0,C 180,E1 -17862.538,E2 -17862.538} C_VEL
LIN {X 0,Y 270.225,Z 283.636,A -85,B 0,C 180,E1 -17866.732,E2 -17866.732} C_VEL
LIN {X 0,Y 270.241,Z 283.634,A -85,B 0,C 180,E1 -17869.444,E2 -17869.444} C_VEL
LIN {X 0,Y 270.247,Z 283.632,A -85,B 0,C 180,E1 -17873.718,E2 -17873.718} C_VEL
LIN {X 0,Y 270.194,Z 283.643,A -85,B 0,C 180,E1 -17876.889,E2 -17876.889} C_VEL
LIN {X 0,Y 270.218,Z 283.637,A -85,B 0,C 180,E1 -17880.383,E2 -17880.383} C_VEL
LIN {X 0,Y 270.252,Z 283.631,A -85,B 0,C 180,E1 -17883.761,E2 -17883.761} C_VEL
LIN {X 0,Y 270.217,Z 283.637,A -85,B 0,C 180,E1 -17887.036,E2 -17887.036} C_VEL
LIN {X 0,Y 270.183,Z 283.643,A -85,B 0,C 180,E1 -17890.234,E2 -17890.234} C_VEL
LIN {X 0,Y 269.884,Z 283.681,A -85,B 0,C 180,E1 -17894.46,E2 -17894.46} C_VEL
LIN {X 0,Y 269.404,Z 283.889,A -85,B 0,C 180,E1 -17897.761,E2 -17897.761} C_VEL
LIN {X 0,Y 269.388,Z 288.11,A -85,B 0,C 180,E1 -17902.503,E2 -17902.503} C_VEL
LIN {X 0,Y 269.2,Z 290.791,A -85,B 0,C 180,E1 -17905.412,E2 -17905.412} C_VEL
LIN {X 0,Y 271.119,Z 301.671,A -85,B 0,C 180,E1 -17906.189,E2 -17906.189} C_VEL
LIN {X 0,Y 272.314,Z 310.859,A -85,B 0,C 180,E1 -17907.039,E2 -17907.039} C_VEL
LIN {X 0,Y 273.144,Z 317.517,A -85,B 0,C 180,E1 -17907.786,E2 -17907.786} C_VEL
LIN {X 0,Y 272.4,Z 326.1,A -85,B 0,C 180,E1 -17908.889,E2 -17908.889} C_VEL
LIN {X 0,Y 271.582,Z 334.191,A -85,B 0,C 180,E1 -17910.183,E2 -17910.183} C_VEL
LIN {X 0,Y 270.866,Z 340.869,A -85,B 0,C 180,E1 -17911.485,E2 -17911.485} C_VEL
LIN {X 0,Y 270.204,Z 347.196,A -85,B 0,C 180,E1 -17912.98,E2 -17912.98} C_VEL
LIN {X 0,Y 269.594,Z 352.464,A -85,B 0,C 180,E1 -17914.483,E2 -17914.483} C_VEL
LIN {X 0,Y 269.278,Z 356.833,A -85,B 0,C 180,E1 -17915.99,E2 -17915.99} C_VEL
LIN {X 0,Y 268.85,Z 360.488,A -85,B 0,C 180,E1 -17917.508,E2 -17917.508} C_VEL
LIN {X 0,Y 268.569,Z 363.482,A -85,B 0,C 180,E1 -17919.031,E2 -17919.031} C_VEL
LIN {X 0,Y 268.302,Z 365.839,A -85,B 0,C 180,E1 -17920.563,E2 -17920.563} C_VEL
LIN {X 0,Y 268.198,Z 367.561,A -85,B 0,C 180,E1 -17922.099,E2 -17922.099} C_VEL
LIN {X 0,Y 268.207,Z 369.124,A -85,B 0,C 180,E1 -17924.195,E2 -17924.195} C_VEL
LIN {X 0,Y 268.385,Z 369.678,A -85,B 0,C 180,E1 -17926.739,E2 -17926.739} C_VEL
LIN {X 0,Y 268.668,Z 369.36,A -85,B 0,C 180,E1 -17928.292,E2 -17928.292} C_VEL
LIN {X 0,Y 269.099,Z 368.384,A -85,B 0,C 180,E1 -17929.926,E2 -17929.926} C_VEL
LIN {X 0,Y 269.875,Z 366.11,A -85,B 0,C 180,E1 -17932.183,E2 -17932.183} C_VEL
LIN {X 0,Y 270.964,Z 362.328,A -85,B 0,C 180,E1 -17934.516,E2 -17934.516} C_VEL
LIN {X 0,Y 272.43,Z 357.067,A -85,B 0,C 180,E1 -17936.835,E2 -17936.835} C_VEL
LIN {X 0,Y 273.903,Z 351.346,A -85,B 0,C 180,E1 -17938.755,E2 -17938.755} C_VEL
LIN {X 0,Y 275.622,Z 343.977,A -85,B 0,C 180,E1 -17940.66,E2 -17940.66} C_VEL
LIN {X 0,Y 277.215,Z 336.548,A -85,B 0,C 180,E1 -17942.165,E2 -17942.165} C_VEL
LIN {X 0,Y 278.571,Z 329.894,A -85,B 0,C 180,E1 -17943.269,E2 -17943.269} C_VEL
LIN {X 0,Y 278.735,Z 327.186,A -85,B 0,C 180,E1 -17943.696,E2 -17943.696} C_VEL
LIN {X 0,Y 277.293,Z 317.838,A -85,B 0,C 180,E1 -17945.183,E2 -17945.183} C_VEL
LIN {X 0,Y 274.602,Z 306.969,A -85,B 0,C 180,E1 -17946.652,E2 -17946.652} C_VEL
LIN {X 0,Y 271.518,Z 297.465,A -85,B 0,C 180,E1 -17947.763,E2 -17947.763} C_VEL
LIN {X 0,Y 269.656,Z 291.789,A -85,B 0,C 180,E1 -17948.357,E2 -17948.357} C_VEL
LIN {X 0,Y 270.025,Z 288.45,A -85,B 0,C 180,E1 -17952.584,E2 -17952.584} C_VEL
LIN {X 0,Y 270.18,Z 286.332,A -85,B 0,C 180,E1 -17955.391,E2 -17955.391} C_VEL
LIN {X 0,Y 270.139,Z 283.796,A -85,B 0,C 180,E1 -17958.976,E2 -17958.976} C_VEL
LIN {X 0,Y 270.189,Z 283.647,A -85,B 0,C 180,E1 -17961.375,E2 -17961.375} C_VEL
LIN {X 0,Y 270.197,Z 283.644,A -85,B 0,C 180,E1 -17965.098,E2 -17965.098} C_VEL
LIN {X 0,Y 270.183,Z 283.642,A -85,B 0,C 180,E1 -17969.132,E2 -17969.132} C_VEL
LIN {X 0,Y 270.247,Z 283.636,A -85,B 0,C 180,E1 -17972.148,E2 -17972.148} C_VEL
LIN {X 0,Y 270.221,Z 283.636,A -85,B 0,C 180,E1 -17975.54,E2 -17975.54} C_VEL
LIN {X 0,Y 270.286,Z 283.63,A -85,B 0,C 180,E1 -17980.247,E2 -17980.247} C_VEL
LIN {X 0,Y 270.389,Z 283.614,A -85,B 0,C 180,E1 -17984.938,E2 -17984.938} C_VEL
LIN {X 0,Y 270.4,Z 283.61,A -85,B 0,C 180,E1 -17989.52,E2 -17989.52} C_VEL
LIN {X 0,Y 270.558,Z 283.595,A -85,B 0,C 180,E1 -17992.54,E2 -17992.54} C_VEL
LIN {X 0,Y 270.778,Z 283.564,A -85,B 0,C 180,E1 -17998.515,E2 -17998.515} C_VEL
LIN {X 0,Y 270.776,Z 283.564,A -85,B 0,C 180,E1 -18001.49,E2 -18001.49} C_VEL
LIN {X 0,Y 270.602,Z 283.591,A -85,B 0,C 180,E1 -18007.464,E2 -18007.464} C_VEL
LIN {X 0,Y 270.434,Z 283.612,A -85,B 0,C 180,E1 -18010.484,E2 -18010.484} C_VEL
LIN {X 0,Y 270.396,Z 283.616,A -85,B 0,C 180,E1 -18015.067,E2 -18015.067} C_VEL
LIN {X 0,Y 270.284,Z 283.63,A -85,B 0,C 180,E1 -18019.597,E2 -18019.597} C_VEL
LIN {X 0,Y 269.66,Z 283.714,A -85,B 0,C 180,E1 -18020.84,E2 -18020.84} C_VEL
LIN {X 0,Y 266.771,Z 284.073,A -85,B 0,C 180,E1 -18022.864,E2 -18022.864} C_VEL
LIN {X 0,Y 264.281,Z 284.382,A -85,B 0,C 180,E1 -18024.51,E2 -18024.51} C_VEL
LIN {X 0,Y 263.207,Z 284.515,A -85,B 0,C 180,E1 -18025.788,E2 -18025.788} C_VEL
LIN {X 0,Y 263.12,Z 284.522,A -85,B 0,C 180,E1 -18026.221,E2 -18026.221} C_VEL
LIN {X 0,Y 263.129,Z 284.526,A -85,B 0,C 180,E1 -18028.738,E2 -18028.738} C_VEL
LIN {X 0,Y 263.124,Z 284.529,A -85,B 0,C 180,E1 -18032.292,E2 -18032.292} C_VEL
LIN {X 0,Y 263.185,Z 284.52,A -85,B 0,C 180,E1 -18035.981,E2 -18035.981} C_VEL
LIN {X 0,Y 263.154,Z 284.534,A -85,B 0,C 180,E1 -18039.866,E2 -18039.866} C_VEL
LIN {X 0,Y 263.767,Z 288.107,A -85,B 0,C 180,E1 -18043.998,E2 -18043.998} C_VEL
LIN {X 0,Y 264.497,Z 292.334,A -85,B 0,C 180,E1 -18048.376,E2 -18048.376} C_VEL
LIN {X 0,Y 265.289,Z 296.81,A -85,B 0,C 180,E1 -18052.635,E2 -18052.635} C_VEL
LIN {X 0,Y 265.586,Z 299.619,A -85,B 0,C 180,E1 -18055.121,E2 -18055.121} C_VEL
LIN {X 0,Y 265.411,Z 302.043,A -85,B 0,C 180,E1 -18057.126,E2 -18057.126} C_VEL
LIN {X 0,Y 264.163,Z 307.474,A -85,B 0,C 180,E1 -18061.4,E2 -18061.4} C_VEL
LIN {X 0,Y 263.256,Z 312.058,A -85,B 0,C 180,E1 -18064.861,E2 -18064.861} C_VEL
LIN {X 0,Y 266.448,Z 325.624,A -85,B 0,C 180,E1 -18066.182,E2 -18066.182} C_VEL
LIN {X 0,Y 268.034,Z 334.682,A -85,B 0,C 180,E1 -18067.232,E2 -18067.232} C_VEL
LIN {X 0,Y 268.957,Z 342.955,A -85,B 0,C 180,E1 -18068.334,E2 -18068.334} C_VEL
LIN {X 0,Y 269.331,Z 351.059,A -85,B 0,C 180,E1 -18069.576,E2 -18069.576} C_VEL
LIN {X 0,Y 269.157,Z 357.974,A -85,B 0,C 180,E1 -18070.79,E2 -18070.79} C_VEL
LIN {X 0,Y 268.089,Z 364.458,A -85,B 0,C 180,E1 -18072.062,E2 -18072.062} C_VEL
LIN {X 0,Y 266.465,Z 370.82,A -85,B 0,C 180,E1 -18073.531,E2 -18073.531} C_VEL
LIN {X 0,Y 264.801,Z 377.297,A -85,B 0,C 180,E1 -18075.398,E2 -18075.398} C_VEL
LIN {X 0,Y 263.779,Z 381.523,A -85,B 0,C 180,E1 -18076.913,E2 -18076.913} C_VEL
LIN {X 0,Y 262.867,Z 385.044,A -85,B 0,C 180,E1 -18078.435,E2 -18078.435} C_VEL
LIN {X 0,Y 261.915,Z 389.117,A -85,B 0,C 180,E1 -18080.737,E2 -18080.737} C_VEL
LIN {X 0,Y 261.496,Z 391.127,A -85,B 0,C 180,E1 -18082.279,E2 -18082.279} C_VEL
LIN {X 0,Y 261.163,Z 393.207,A -85,B 0,C 180,E1 -18084.692,E2 -18084.692} C_VEL
LIN {X 0,Y 261.182,Z 394.06,A -85,B 0,C 180,E1 -18086.917,E2 -18086.917} C_VEL
LIN {X 0,Y 261.202,Z 394.014,A -85,B 0,C 180,E1 -18088.46,E2 -18088.46} C_VEL
LIN {X 0,Y 261.252,Z 393.508,A -85,B 0,C 180,E1 -18090.002,E2 -18090.002} C_VEL
LIN {X 0,Y 261.238,Z 392.513,A -85,B 0,C 180,E1 -18091.544,E2 -18091.544} C_VEL
LIN {X 0,Y 261.249,Z 389.889,A -85,B 0,C 180,E1 -18093.858,E2 -18093.858} C_VEL
LIN {X 0,Y 261.214,Z 387.455,A -85,B 0,C 180,E1 -18095.428,E2 -18095.428} C_VEL
LIN {X 0,Y 261.519,Z 382.586,A -85,B 0,C 180,E1 -18097.724,E2 -18097.724} C_VEL
LIN {X 0,Y 261.818,Z 378.469,A -85,B 0,C 180,E1 -18099.27,E2 -18099.27} C_VEL
LIN {X 0,Y 262.245,Z 373.502,A -85,B 0,C 180,E1 -18100.814,E2 -18100.814} C_VEL
LIN {X 0,Y 262.835,Z 367.507,A -85,B 0,C 180,E1 -18102.354,E2 -18102.354} C_VEL
LIN {X 0,Y 263.6,Z 360.203,A -85,B 0,C 180,E1 -18103.886,E2 -18103.886} C_VEL
LIN {X 0,Y 264.38,Z 353.648,A -85,B 0,C 180,E1 -18105.024,E2 -18105.024} C_VEL
LIN {X 0,Y 264.25,Z 345.654,A -85,B 0,C 180,E1 -18106.2,E2 -18106.2} C_VEL
LIN {X 0,Y 263.861,Z 337.023,A -85,B 0,C 180,E1 -18107.238,E2 -18107.238} C_VEL
LIN {X 0,Y 263.29,Z 328.29,A -85,B 0,C 180,E1 -18108.08,E2 -18108.08} C_VEL
LIN {X 0,Y 262.357,Z 318.682,A -85,B 0,C 180,E1 -18108.796,E2 -18108.796} C_VEL
LIN {X 0,Y 261.725,Z 313.06,A -85,B 0,C 180,E1 -18109.143,E2 -18109.143} C_VEL
LIN {X 0,Y 262.379,Z 306.633,A -85,B 0,C 180,E1 -18113.692,E2 -18113.692} C_VEL
LIN {X 0,Y 263.301,Z 300.25,A -85,B 0,C 180,E1 -18118.253,E2 -18118.253} C_VEL
LIN {X 0,Y 264.488,Z 293.774,A -85,B 0,C 180,E1 -18123.008,E2 -18123.008} C_VEL
LIN {X 0,Y 264.309,Z 290.201,A -85,B 0,C 180,E1 -18125.804,E2 -18125.804} C_VEL
LIN {X 0,Y 263.267,Z 284.505,A -85,B 0,C 180,E1 -18130.534,E2 -18130.534} C_VEL
LIN {X 0,Y 263.134,Z 284.522,A -85,B 0,C 180,E1 -18133.984,E2 -18133.984} C_VEL
LIN {X 0,Y 263.136,Z 284.519,A -85,B 0,C 180,E1 -18138.406,E2 -18138.406} C_VEL
LIN {X 0,Y 263.194,Z 284.51,A -85,B 0,C 180,E1 -18143.236,E2 -18143.236} C_VEL
LIN {X 0,Y 263.144,Z 284.518,A -85,B 0,C 180,E1 -18147.711,E2 -18147.711} C_VEL
LIN {X 0,Y 263.213,Z 284.51,A -85,B 0,C 180,E1 -18151.782,E2 -18151.782} C_VEL
LIN {X 0,Y 263.212,Z 284.511,A -85,B 0,C 180,E1 -18155.211,E2 -18155.211} C_VEL
LIN {X 0,Y 263.246,Z 284.504,A -85,B 0,C 180,E1 -18159.689,E2 -18159.689} C_VEL
LIN {X 0,Y 263.32,Z 284.496,A -85,B 0,C 180,E1 -18164.518,E2 -18164.518} C_VEL
LIN {X 0,Y 263.355,Z 284.491,A -85,B 0,C 180,E1 -18169.231,E2 -18169.231} C_VEL
LIN {X 0,Y 263.552,Z 284.467,A -85,B 0,C 180,E1 -18172.335,E2 -18172.335} C_VEL
LIN {X 0,Y 263.758,Z 284.441,A -85,B 0,C 180,E1 -18178.47,E2 -18178.47} C_VEL
LIN {X 0,Y 263.759,Z 284.439,A -85,B 0,C 180,E1 -18181.524,E2 -18181.524} C_VEL
LIN {X 0,Y 263.578,Z 284.462,A -85,B 0,C 180,E1 -18187.658,E2 -18187.658} C_VEL
LIN {X 0,Y 263.379,Z 284.485,A -85,B 0,C 180,E1 -18190.762,E2 -18190.762} C_VEL
LIN {X 0,Y 263.348,Z 284.492,A -85,B 0,C 180,E1 -18195.475,E2 -18195.475} C_VEL
LIN {X 0,Y 263.266,Z 284.5,A -85,B 0,C 180,E1 -18200.303,E2 -18200.303} C_VEL
LIN {X 0,Y 263.209,Z 284.509,A -85,B 0,C 180,E1 -18205.288,E2 -18205.288} C_VEL
LIN {X 0,Y 263.174,Z 284.513,A -85,B 0,C 180,E1 -18208.726,E2 -18208.726} C_VEL
LIN {X 0,Y 263.131,Z 284.519,A -85,B 0,C 180,E1 -18212.284,E2 -18212.284} C_VEL
LIN {X 0,Y 263.187,Z 284.513,A -85,B 0,C 180,E1 -18215.974,E2 -18215.974} C_VEL
LIN {X 0,Y 263.189,Z 284.512,A -85,B 0,C 180,E1 -18219.853,E2 -18219.853} C_VEL
LIN {X 0,Y 263.185,Z 284.512,A -85,B 0,C 180,E1 -18223.966,E2 -18223.966} C_VEL
LIN {X 0,Y 263.205,Z 284.509,A -85,B 0,C 180,E1 -18228.381,E2 -18228.381} C_VEL
LIN {X 0,Y 263.195,Z 284.513,A -85,B 0,C 180,E1 -18233.227,E2 -18233.227} C_VEL
LIN {X 0,Y 263.175,Z 284.513,A -85,B 0,C 180,E1 -18235.887,E2 -18235.887} C_VEL
LIN {X 0,Y 263.14,Z 284.518,A -85,B 0,C 180,E1 -18239.503,E2 -18239.503} C_VEL
LIN {X 0,Y 263.182,Z 284.515,A -85,B 0,C 180,E1 -18243,E2 -18243} C_VEL
LIN {X 0,Y 263.171,Z 284.516,A -85,B 0,C 180,E1 -18246.384,E2 -18246.384} C_VEL
LIN {X 0,Y 263.189,Z 284.512,A -85,B 0,C 180,E1 -18249.685,E2 -18249.685} C_VEL
LIN {X 0,Y 262.848,Z 284.557,A -85,B 0,C 180,E1 -18254.49,E2 -18254.49} C_VEL
LIN {X 0,Y 262.367,Z 284.731,A -85,B 0,C 180,E1 -18257.82,E2 -18257.82} C_VEL
LIN {X 0,Y 262.332,Z 288.731,A -85,B 0,C 180,E1 -18262.384,E2 -18262.384} C_VEL
LIN {X 0,Y 262.146,Z 291.291,A -85,B 0,C 180,E1 -18265.048,E2 -18265.048} C_VEL
LIN {X 0,Y 264.214,Z 302.726,A -85,B 0,C 180,E1 -18265.899,E2 -18265.899} C_VEL
LIN {X 0,Y 265.374,Z 311.756,A -85,B 0,C 180,E1 -18266.772,E2 -18266.772} C_VEL
LIN {X 0,Y 266.181,Z 318.303,A -85,B 0,C 180,E1 -18267.539,E2 -18267.539} C_VEL
LIN {X 0,Y 265.422,Z 326.801,A -85,B 0,C 180,E1 -18268.67,E2 -18268.67} C_VEL
LIN {X 0,Y 264.649,Z 333.814,A -85,B 0,C 180,E1 -18269.808,E2 -18269.808} C_VEL
LIN {X 0,Y 263.943,Z 340.599,A -85,B 0,C 180,E1 -18271.142,E2 -18271.142} C_VEL
LIN {X 0,Y 263.214,Z 347.031,A -85,B 0,C 180,E1 -18272.676,E2 -18272.676} C_VEL
LIN {X 0,Y 262.609,Z 352.379,A -85,B 0,C 180,E1 -18274.219,E2 -18274.219} C_VEL
LIN {X 0,Y 262.336,Z 355.853,A -85,B 0,C 180,E1 -18275.378,E2 -18275.378} C_VEL
LIN {X 0,Y 261.915,Z 359.653,A -85,B 0,C 180,E1 -18276.901,E2 -18276.901} C_VEL
LIN {X 0,Y 261.427,Z 364.199,A -85,B 0,C 180,E1 -18279.28,E2 -18279.28} C_VEL
LIN {X 0,Y 261.172,Z 366.494,A -85,B 0,C 180,E1 -18280.855,E2 -18280.855} C_VEL
LIN {X 0,Y 261.116,Z 368.164,A -85,B 0,C 180,E1 -18282.432,E2 -18282.432} C_VEL
LIN {X 0,Y 261.118,Z 369.46,A -85,B 0,C 180,E1 -18284.333,E2 -18284.333} C_VEL
LIN {X 0,Y 261.356,Z 369.962,A -85,B 0,C 180,E1 -18287.203,E2 -18287.203} C_VEL
LIN {X 0,Y 261.705,Z 369.57,A -85,B 0,C 180,E1 -18288.797,E2 -18288.797} C_VEL
LIN {X 0,Y 262.166,Z 368.605,A -85,B 0,C 180,E1 -18290.393,E2 -18290.393} C_VEL
LIN {X 0,Y 263.048,Z 366.074,A -85,B 0,C 180,E1 -18292.791,E2 -18292.791} C_VEL
LIN {X 0,Y 263.815,Z 363.687,A -85,B 0,C 180,E1 -18294.386,E2 -18294.386} C_VEL
LIN {X 0,Y 265.267,Z 358.722,A -85,B 0,C 180,E1 -18296.767,E2 -18296.767} C_VEL
LIN {X 0,Y 266.48,Z 354.519,A -85,B 0,C 180,E1 -18298.339,E2 -18298.339} C_VEL
LIN {X 0,Y 267.781,Z 349.084,A -85,B 0,C 180,E1 -18299.999,E2 -18299.999} C_VEL
LIN {X 0,Y 269.296,Z 343.161,A -85,B 0,C 180,E1 -18301.461,E2 -18301.461} C_VEL
LIN {X 0,Y 270.743,Z 336.562,A -85,B 0,C 180,E1 -18302.809,E2 -18302.809} C_VEL
LIN {X 0,Y 272.153,Z 329.37,A -85,B 0,C 180,E1 -18304.017,E2 -18304.017} C_VEL
LIN {X 0,Y 271.147,Z 321.988,A -85,B 0,C 180,E1 -18305.284,E2 -18305.284} C_VEL
LIN {X 0,Y 269.666,Z 314.473,A -85,B 0,C 180,E1 -18306.429,E2 -18306.429} C_VEL
LIN {X 0,Y 267.317,Z 305.841,A -85,B 0,C 180,E1 -18307.605,E2 -18307.605} C_VEL
LIN {X 0,Y 264.274,Z 296.906,A -85,B 0,C 180,E1 -18308.688,E2 -18308.688} C_VEL
LIN {X 0,Y 262.666,Z 292.174,A -85,B 0,C 180,E1 -18309.21,E2 -18309.21} C_VEL
LIN {X 0,Y 262.94,Z 290.075,A -85,B 0,C 180,E1 -18311.926,E2 -18311.926} C_VEL
LIN {X 0,Y 263.096,Z 288.514,A -85,B 0,C 180,E1 -18313.987,E2 -18313.987} C_VEL
LIN {X 0,Y 263.195,Z 286.97,A -85,B 0,C 180,E1 -18316.131,E2 -18316.131} C_VEL
LIN {X 0,Y 263.129,Z 285.397,A -85,B 0,C 180,E1 -18318.402,E2 -18318.402} C_VEL
LIN {X 0,Y 263.07,Z 284.529,A -85,B 0,C 180,E1 -18320.126,E2 -18320.126} C_VEL
LIN {X 0,Y 263.169,Z 284.52,A -85,B 0,C 180,E1 -18324.023,E2 -18324.023} C_VEL
LIN {X 0,Y 263.116,Z 284.523,A -85,B 0,C 180,E1 -18327.713,E2 -18327.713} C_VEL
LIN {X 0,Y 263.179,Z 284.514,A -85,B 0,C 180,E1 -18331.787,E2 -18331.787} C_VEL
LIN {X 0,Y 263.185,Z 284.515,A -85,B 0,C 180,E1 -18335.214,E2 -18335.214} C_VEL
LIN {X 0,Y 263.248,Z 284.503,A -85,B 0,C 180,E1 -18339.696,E2 -18339.696} C_VEL
LIN {X 0,Y 263.337,Z 284.496,A -85,B 0,C 180,E1 -18344.524,E2 -18344.524} C_VEL
LIN {X 0,Y 263.342,Z 284.49,A -85,B 0,C 180,E1 -18349.236,E2 -18349.236} C_VEL
LIN {X 0,Y 263.52,Z 284.473,A -85,B 0,C 180,E1 -18352.34,E2 -18352.34} C_VEL
LIN {X 0,Y 263.742,Z 284.44,A -85,B 0,C 180,E1 -18358.476,E2 -18358.476} C_VEL
LIN {X 0,Y 263.741,Z 284.44,A -85,B 0,C 180,E1 -18361.53,E2 -18361.53} C_VEL
LIN {X 0,Y 263.564,Z 284.468,A -85,B 0,C 180,E1 -18367.664,E2 -18367.664} C_VEL
LIN {X 0,Y 263.366,Z 284.491,A -85,B 0,C 180,E1 -18370.768,E2 -18370.768} C_VEL
LIN {X 0,Y 263.344,Z 284.495,A -85,B 0,C 180,E1 -18375.481,E2 -18375.481} C_VEL
LIN {X 0,Y 263.256,Z 284.505,A -85,B 0,C 180,E1 -18380.31,E2 -18380.31} C_VEL
LIN {X 0,Y 263.163,Z 284.519,A -85,B 0,C 180,E1 -18385.298,E2 -18385.298} C_VEL
LIN {X 0,Y 263.12,Z 284.522,A -85,B 0,C 180,E1 -18386.221,E2 -18386.221} C_VEL
LIN {X 0,Y 262.439,Z 284.613,A -85,B 0,C 180,E1 -18387.498,E2 -18387.498} C_VEL
LIN {X 0,Y 259.553,Z 284.973,A -85,B 0,C 180,E1 -18389.577,E2 -18389.577} C_VEL
LIN {X 0,Y 257.131,Z 285.275,A -85,B 0,C 180,E1 -18391.269,E2 -18391.269} C_VEL
LIN {X 0,Y 256.127,Z 285.4,A -85,B 0,C 180,E1 -18392.581,E2 -18392.581} C_VEL
LIN {X 0,Y 256.064,Z 285.407,A -85,B 0,C 180,E1 -18393.026,E2 -18393.026} C_VEL
LIN {X 0,Y 256.137,Z 285.397,A -85,B 0,C 180,E1 -18397.281,E2 -18397.281} C_VEL
LIN {X 0,Y 256.116,Z 285.489,A -85,B 0,C 180,E1 -18399.137,E2 -18399.137} C_VEL
LIN {X 0,Y 256.676,Z 288.878,A -85,B 0,C 180,E1 -18403.201,E2 -18403.201} C_VEL
LIN {X 0,Y 257.331,Z 292.842,A -85,B 0,C 180,E1 -18407.513,E2 -18407.513} C_VEL
LIN {X 0,Y 258.05,Z 296.554,A -85,B 0,C 180,E1 -18411.218,E2 -18411.218} C_VEL
LIN {X 0,Y 258.575,Z 300.214,A -85,B 0,C 180,E1 -18414.629,E2 -18414.629} C_VEL
LIN {X 0,Y 258.394,Z 303.015,A -85,B 0,C 180,E1 -18417.048,E2 -18417.048} C_VEL
LIN {X 0,Y 257.215,Z 307.866,A -85,B 0,C 180,E1 -18420.972,E2 -18420.972} C_VEL
LIN {X 0,Y 256.377,Z 311.715,A -85,B 0,C 180,E1 -18423.988,E2 -18423.988} C_VEL
LIN {X 0,Y 258.589,Z 320.67,A -85,B 0,C 180,E1 -18424.846,E2 -18424.846} C_VEL
LIN {X 0,Y 261.053,Z 332.882,A -85,B 0,C 180,E1 -18426.258,E2 -18426.258} C_VEL
LIN {X 0,Y 262.201,Z 342.17,A -85,B 0,C 180,E1 -18427.53,E2 -18427.53} C_VEL
LIN {X 0,Y 262.615,Z 350.389,A -85,B 0,C 180,E1 -18428.824,E2 -18428.824} C_VEL
LIN {X 0,Y 262.448,Z 358.036,A -85,B 0,C 180,E1 -18430.214,E2 -18430.214} C_VEL
LIN {X 0,Y 261.784,Z 363.013,A -85,B 0,C 180,E1 -18431.209,E2 -18431.209} C_VEL
LIN {X 0,Y 260.061,Z 369.555,A -85,B 0,C 180,E1 -18432.709,E2 -18432.709} C_VEL
LIN {X 0,Y 258.571,Z 375.015,A -85,B 0,C 180,E1 -18434.231,E2 -18434.231} C_VEL
LIN {X 0,Y 257.356,Z 379.594,A -85,B 0,C 180,E1 -18435.775,E2 -18435.775} C_VEL
LIN {X 0,Y 256.365,Z 383.405,A -85,B 0,C 180,E1 -18437.334,E2 -18437.334} C_VEL
LIN {X 0,Y 255.184,Z 387.809,A -85,B 0,C 180,E1 -18439.69,E2 -18439.69} C_VEL
LIN {X 0,Y 254.432,Z 390.93,A -85,B 0,C 180,E1 -18442.064,E2 -18442.064} C_VEL
LIN {X 0,Y 254.06,Z 393.12,A -85,B 0,C 180,E1 -18444.803,E2 -18444.803} C_VEL
LIN {X 0,Y 254.092,Z 393.756,A -85,B 0,C 180,E1 -18446.831,E2 -18446.831} C_VEL
LIN {X 0,Y 254.127,Z 393.658,A -85,B 0,C 180,E1 -18448.417,E2 -18448.417} C_VEL
LIN {X 0,Y 254.174,Z 393.098,A -85,B 0,C 180,E1 -18450.002,E2 -18450.002} C_VEL
LIN {X 0,Y 254.165,Z 392.059,A -85,B 0,C 180,E1 -18451.587,E2 -18451.587} C_VEL
LIN {X 0,Y 254.168,Z 389.366,A -85,B 0,C 180,E1 -18453.966,E2 -18453.966} C_VEL
LIN {X 0,Y 254.142,Z 387.218,A -85,B 0,C 180,E1 -18455.396,E2 -18455.396} C_VEL
LIN {X 0,Y 254.347,Z 383.834,A -85,B 0,C 180,E1 -18457.145,E2 -18457.145} C_VEL
LIN {X 0,Y 254.783,Z 377.743,A -85,B 0,C 180,E1 -18459.529,E2 -18459.529} C_VEL
LIN {X 0,Y 255.231,Z 372.693,A -85,B 0,C 180,E1 -18461.115,E2 -18461.115} C_VEL
LIN {X 0,Y 255.855,Z 366.602,A -85,B 0,C 180,E1 -18462.696,E2 -18462.696} C_VEL
LIN {X 0,Y 256.708,Z 359.189,A -85,B 0,C 180,E1 -18464.266,E2 -18464.266} C_VEL
LIN {X 0,Y 257.424,Z 352.478,A -85,B 0,C 180,E1 -18465.439,E2 -18465.439} C_VEL
LIN {X 0,Y 257.172,Z 344.541,A -85,B 0,C 180,E1 -18466.622,E2 -18466.622} C_VEL
LIN {X 0,Y 256.753,Z 335.366,A -85,B 0,C 180,E1 -18467.731,E2 -18467.731} C_VEL
LIN {X 0,Y 256.036,Z 324.96,A -85,B 0,C 180,E1 -18468.714,E2 -18468.714} C_VEL
LIN {X 0,Y 254.687,Z 312.727,A -85,B 0,C 180,E1 -18469.545,E2 -18469.545} C_VEL
LIN {X 0,Y 255.428,Z 306.131,A -85,B 0,C 180,E1 -18474.378,E2 -18474.378} C_VEL
LIN {X 0,Y 256.299,Z 300.345,A -85,B 0,C 180,E1 -18478.657,E2 -18478.657} C_VEL
LIN {X 0,Y 257.453,Z 294.503,A -85,B 0,C 180,E1 -18483.093,E2 -18483.093} C_VEL
LIN {X 0,Y 257.219,Z 290.881,A -85,B 0,C 180,E1 -18485.978,E2 -18485.978} C_VEL
LIN {X 0,Y 256.212,Z 285.383,A -85,B 0,C 180,E1 -18490.816,E2 -18490.816} C_VEL
LIN {X 0,Y 256.069,Z 285.399,A -85,B 0,C 180,E1 -18495.53,E2 -18495.53} C_VEL
LIN {X 0,Y 256.066,Z 285.399,A -85,B 0,C 180,E1 -18498.796,E2 -18498.796} C_VEL
LIN {X 0,Y 256.142,Z 285.388,A -85,B 0,C 180,E1 -18502.867,E2 -18502.867} C_VEL
LIN {X 0,Y 256.079,Z 285.397,A -85,B 0,C 180,E1 -18506.706,E2 -18506.706} C_VEL
LIN {X 0,Y 256.126,Z 285.389,A -85,B 0,C 180,E1 -18510.399,E2 -18510.399} C_VEL
LIN {X 0,Y 256.182,Z 285.385,A -85,B 0,C 180,E1 -18514.869,E2 -18514.869} C_VEL
LIN {X 0,Y 256.158,Z 285.387,A -85,B 0,C 180,E1 -18519.102,E2 -18519.102} C_VEL
LIN {X 0,Y 256.24,Z 285.377,A -85,B 0,C 180,E1 -18524.079,E2 -18524.079} C_VEL
LIN {X 0,Y 256.297,Z 285.369,A -85,B 0,C 180,E1 -18528.931,E2 -18528.931} C_VEL
LIN {X 0,Y 256.513,Z 285.343,A -85,B 0,C 180,E1 -18532.124,E2 -18532.124} C_VEL
LIN {X 0,Y 256.504,Z 285.344,A -85,B 0,C 180,E1 -18536.856,E2 -18536.856} C_VEL
LIN {X 0,Y 256.765,Z 285.308,A -85,B 0,C 180,E1 -18539.997,E2 -18539.997} C_VEL
LIN {X 0,Y 256.506,Z 285.344,A -85,B 0,C 180,E1 -18543.138,E2 -18543.138} C_VEL
LIN {X 0,Y 256.546,Z 285.339,A -85,B 0,C 180,E1 -18547.87,E2 -18547.87} C_VEL
LIN {X 0,Y 256.314,Z 285.364,A -85,B 0,C 180,E1 -18551.063,E2 -18551.063} C_VEL
LIN {X 0,Y 256.298,Z 285.372,A -85,B 0,C 180,E1 -18555.912,E2 -18555.912} C_VEL
LIN {X 0,Y 256.169,Z 285.382,A -85,B 0,C 180,E1 -18560.891,E2 -18560.891} C_VEL
LIN {X 0,Y 256.189,Z 285.383,A -85,B 0,C 180,E1 -18565.135,E2 -18565.135} C_VEL
LIN {X 0,Y 256.11,Z 285.396,A -85,B 0,C 180,E1 -18569.596,E2 -18569.596} C_VEL
LIN {X 0,Y 256.083,Z 285.399,A -85,B 0,C 180,E1 -18573.286,E2 -18573.286} C_VEL
LIN {X 0,Y 256.138,Z 285.392,A -85,B 0,C 180,E1 -18577.275,E2 -18577.275} C_VEL
LIN {X 0,Y 256.156,Z 285.389,A -85,B 0,C 180,E1 -18581.179,E2 -18581.179} C_VEL
LIN {X 0,Y 256.111,Z 285.395,A -85,B 0,C 180,E1 -18585.513,E2 -18585.513} C_VEL
LIN {X 0,Y 256.125,Z 285.393,A -85,B 0,C 180,E1 -18588.808,E2 -18588.808} C_VEL
LIN {X 0,Y 256.146,Z 285.392,A -85,B 0,C 180,E1 -18592.868,E2 -18592.868} C_VEL
LIN {X 0,Y 256.076,Z 285.4,A -85,B 0,C 180,E1 -18596.706,E2 -18596.706} C_VEL
LIN {X 0,Y 256.127,Z 285.391,A -85,B 0,C 180,E1 -18601.401,E2 -18601.401} C_VEL
LIN {X 0,Y 256.155,Z 285.387,A -85,B 0,C 180,E1 -18605.696,E2 -18605.696} C_VEL
LIN {X 0,Y 256.117,Z 285.394,A -85,B 0,C 180,E1 -18609.099,E2 -18609.099} C_VEL
LIN {X 0,Y 255.923,Z 285.418,A -85,B 0,C 180,E1 -18612.416,E2 -18612.416} C_VEL
LIN {X 0,Y 255.624,Z 285.454,A -85,B 0,C 180,E1 -18615.672,E2 -18615.672} C_VEL
LIN {X 0,Y 255.308,Z 285.581,A -85,B 0,C 180,E1 -18617.882,E2 -18617.882} C_VEL
LIN {X 0,Y 255.278,Z 289.383,A -85,B 0,C 180,E1 -18622.323,E2 -18622.323} C_VEL
LIN {X 0,Y 255.061,Z 291.412,A -85,B 0,C 180,E1 -18624.612,E2 -18624.612} C_VEL
LIN {X 0,Y 257.163,Z 302.66,A -85,B 0,C 180,E1 -18625.492,E2 -18625.492} C_VEL
LIN {X 0,Y 258.295,Z 310.89,A -85,B 0,C 180,E1 -18626.293,E2 -18626.293} C_VEL
LIN {X 0,Y 259.199,Z 319.097,A -85,B 0,C 180,E1 -18627.278,E2 -18627.278} C_VEL
LIN {X 0,Y 258.416,Z 327.512,A -85,B 0,C 180,E1 -18628.44,E2 -18628.44} C_VEL
LIN {X 0,Y 257.632,Z 334.457,A -85,B 0,C 180,E1 -18629.607,E2 -18629.607} C_VEL
LIN {X 0,Y 257.003,Z 340.335,A -85,B 0,C 180,E1 -18630.781,E2 -18630.781} C_VEL
LIN {X 0,Y 256.261,Z 346.861,A -85,B 0,C 180,E1 -18632.356,E2 -18632.356} C_VEL
LIN {X 0,Y 255.614,Z 352.296,A -85,B 0,C 180,E1 -18633.939,E2 -18633.939} C_VEL
LIN {X 0,Y 255.2,Z 356.822,A -85,B 0,C 180,E1 -18635.529,E2 -18635.529} C_VEL
LIN {X 0,Y 254.74,Z 360.837,A -85,B 0,C 180,E1 -18637.246,E2 -18637.246} C_VEL
LIN {X 0,Y 254.277,Z 364.917,A -85,B 0,C 180,E1 -18639.544,E2 -18639.544} C_VEL
LIN {X 0,Y 254.05,Z 367.102,A -85,B 0,C 180,E1 -18641.163,E2 -18641.163} C_VEL
LIN {X 0,Y 254.005,Z 368.732,A -85,B 0,C 180,E1 -18642.786,E2 -18642.786} C_VEL
LIN {X 0,Y 254.051,Z 369.807,A -85,B 0,C 180,E1 -18644.497,E2 -18644.497} C_VEL
LIN {X 0,Y 254.124,Z 370.248,A -85,B 0,C 180,E1 -18646.053,E2 -18646.053} C_VEL
LIN {X 0,Y 254.346,Z 370.246,A -85,B 0,C 180,E1 -18647.693,E2 -18647.693} C_VEL
LIN {X 0,Y 255.106,Z 369.055,A -85,B 0,C 180,E1 -18650.51,E2 -18650.51} C_VEL
LIN {X 0,Y 255.892,Z 367.1,A -85,B 0,C 180,E1 -18652.611,E2 -18652.611} C_VEL
LIN {X 0,Y 257.05,Z 363.649,A -85,B 0,C 180,E1 -18655.009,E2 -18655.009} C_VEL
LIN {X 0,Y 258.107,Z 360.375,A -85,B 0,C 180,E1 -18656.695,E2 -18656.695} C_VEL
LIN {X 0,Y 259.636,Z 355.284,A -85,B 0,C 180,E1 -18658.713,E2 -18658.713} C_VEL
LIN {X 0,Y 261.137,Z 349.429,A -85,B 0,C 180,E1 -18660.554,E2 -18660.554} C_VEL
LIN {X 0,Y 262.593,Z 344.13,A -85,B 0,C 180,E1 -18661.907,E2 -18661.907} C_VEL
LIN {X 0,Y 264.316,Z 336.599,A -85,B 0,C 180,E1 -18663.483,E2 -18663.483} C_VEL
LIN {X 0,Y 265.513,Z 330.58,A -85,B 0,C 180,E1 -18664.534,E2 -18664.534} C_VEL
LIN {X 0,Y 264.502,Z 322.888,A -85,B 0,C 180,E1 -18665.915,E2 -18665.915} C_VEL
LIN {X 0,Y 262.729,Z 314.316,A -85,B 0,C 180,E1 -18667.275,E2 -18667.275} C_VEL
LIN {X 0,Y 260.331,Z 305.843,A -85,B 0,C 180,E1 -18668.479,E2 -18668.479} C_VEL
LIN {X 0,Y 257.685,Z 298.174,A -85,B 0,C 180,E1 -18669.466,E2 -18669.466} C_VEL
LIN {X 0,Y 255.73,Z 292.561,A -85,B 0,C 180,E1 -18670.116,E2 -18670.116} C_VEL
LIN {X 0,Y 256.015,Z 290.136,A -85,B 0,C 180,E1 -18673.334,E2 -18673.334} C_VEL
LIN {X 0,Y 256.167,Z 287.744,A -85,B 0,C 180,E1 -18676.7,E2 -18676.7} C_VEL
LIN {X 0,Y 256.032,Z 285.448,A -85,B 0,C 180,E1 -18680.224,E2 -18680.224} C_VEL
LIN {X 0,Y 256.126,Z 285.398,A -85,B 0,C 180,E1 -18682.871,E2 -18682.871} C_VEL
LIN {X 0,Y 256.068,Z 285.402,A -85,B 0,C 180,E1 -18686.711,E2 -18686.711} C_VEL
LIN {X 0,Y 256.11,Z 285.394,A -85,B 0,C 180,E1 -18691.412,E2 -18691.412} C_VEL
LIN {X 0,Y 256.127,Z 285.391,A -85,B 0,C 180,E1 -18695.699,E2 -18695.699} C_VEL
LIN {X 0,Y 256.147,Z 285.387,A -85,B 0,C 180,E1 -18699.107,E2 -18699.107} C_VEL
LIN {X 0,Y 256.286,Z 285.374,A -85,B 0,C 180,E1 -18704.087,E2 -18704.087} C_VEL
LIN {X 0,Y 256.282,Z 285.374,A -85,B 0,C 180,E1 -18707.33,E2 -18707.33} C_VEL
LIN {X 0,Y 256.482,Z 285.349,A -85,B 0,C 180,E1 -18712.128,E2 -18712.128} C_VEL
LIN {X 0,Y 256.487,Z 285.346,A -85,B 0,C 180,E1 -18716.861,E2 -18716.861} C_VEL
LIN {X 0,Y 256.755,Z 285.316,A -85,B 0,C 180,E1 -18720.003,E2 -18720.003} C_VEL
LIN {X 0,Y 256.489,Z 285.347,A -85,B 0,C 180,E1 -18723.144,E2 -18723.144} C_VEL
LIN {X 0,Y 256.531,Z 285.344,A -85,B 0,C 180,E1 -18727.876,E2 -18727.876} C_VEL
LIN {X 0,Y 256.302,Z 285.371,A -85,B 0,C 180,E1 -18731.069,E2 -18731.069} C_VEL
LIN {X 0,Y 256.293,Z 285.373,A -85,B 0,C 180,E1 -18735.918,E2 -18735.918} C_VEL
LIN {X 0,Y 256.156,Z 285.391,A -85,B 0,C 180,E1 -18740.899,E2 -18740.899} C_VEL
LIN {X 0,Y 256.128,Z 285.396,A -85,B 0,C 180,E1 -18745.115,E2 -18745.115} C_VEL
LIN {X 0,Y 256.05,Z 285.409,A -85,B 0,C 180,E1 -18749.61,E2 -18749.61} C_VEL
LIN {X 0,Y 256.064,Z 285.407,A -85,B 0,C 180,E1 -18753.026,E2 -18753.026} C_VEL
LIN {X 0,Y 255.432,Z 285.491,A -85,B 0,C 180,E1 -18754.339,E2 -18754.339} C_VEL
LIN {X 0,Y 252.576,Z 285.872,A -85,B 0,C 180,E1 -18756.479,E2 -18756.479} C_VEL
LIN {X 0,Y 250.208,Z 286.573,A -85,B 0,C 180,E1 -18758.215,E2 -18758.215} C_VEL
LIN {X 0,Y 249.304,Z 287.378,A -85,B 0,C 180,E1 -18759.553,E2 -18759.553} C_VEL
LIN {X 0,Y 249.291,Z 287.707,A -85,B 0,C 180,E1 -18760.003,E2 -18760.003} C_VEL
LIN {X 0,Y 249.945,Z 291.61,A -85,B 0,C 180,E1 -18764.667,E2 -18764.667} C_VEL
LIN {X 0,Y 250.67,Z 295.8,A -85,B 0,C 180,E1 -18769.203,E2 -18769.203} C_VEL
LIN {X 0,Y 251.353,Z 299.699,A -85,B 0,C 180,E1 -18773.05,E2 -18773.05} C_VEL
LIN {X 0,Y 251.576,Z 302.937,A -85,B 0,C 180,E1 -18776.036,E2 -18776.036} C_VEL
LIN {X 0,Y 250.529,Z 307.237,A -85,B 0,C 180,E1 -18779.675,E2 -18779.675} C_VEL
LIN {X 0,Y 249.586,Z 311.284,A -85,B 0,C 180,E1 -18782.998,E2 -18782.998} C_VEL
LIN {X 0,Y 251.151,Z 317.647,A -85,B 0,C 180,E1 -18783.663,E2 -18783.663} C_VEL
LIN {X 0,Y 253.229,Z 326.641,A -85,B 0,C 180,E1 -18784.683,E2 -18784.683} C_VEL
LIN {X 0,Y 254.744,Z 335.508,A -85,B 0,C 180,E1 -18785.831,E2 -18785.831} C_VEL
LIN {X 0,Y 255.685,Z 344.41,A -85,B 0,C 180,E1 -18787.149,E2 -18787.149} C_VEL
LIN {X 0,Y 255.943,Z 353.323,A -85,B 0,C 180,E1 -18788.667,E2 -18788.667} C_VEL
LIN {X 0,Y 255.372,Z 361.84,A -85,B 0,C 180,E1 -18790.368,E2 -18790.368} C_VEL
LIN {X 0,Y 253.304,Z 369.718,A -85,B 0,C 180,E1 -18792.232,E2 -18792.232} C_VEL
LIN {X 0,Y 251.754,Z 375.092,A -85,B 0,C 180,E1 -18793.792,E2 -18793.792} C_VEL
LIN {X 0,Y 250.464,Z 379.596,A -85,B 0,C 180,E1 -18795.374,E2 -18795.374} C_VEL
LIN {X 0,Y 249.428,Z 383.364,A -85,B 0,C 180,E1 -18796.975,E2 -18796.975} C_VEL
LIN {X 0,Y 248.198,Z 387.677,A -85,B 0,C 180,E1 -18799.396,E2 -18799.396} C_VEL
LIN {X 0,Y 247.392,Z 390.737,A -85,B 0,C 180,E1 -18801.836,E2 -18801.836} C_VEL
LIN {X 0,Y 246.963,Z 393.005,A -85,B 0,C 180,E1 -18804.904,E2 -18804.904} C_VEL
LIN {X 0,Y 247.007,Z 393.452,A -85,B 0,C 180,E1 -18806.74,E2 -18806.74} C_VEL
LIN {X 0,Y 247.054,Z 393.301,A -85,B 0,C 180,E1 -18808.372,E2 -18808.372} C_VEL
LIN {X 0,Y 247.098,Z 392.688,A -85,B 0,C 180,E1 -18810.002,E2 -18810.002} C_VEL
LIN {X 0,Y 247.093,Z 391.594,A -85,B 0,C 180,E1 -18811.632,E2 -18811.632} C_VEL
LIN {X 0,Y 247.103,Z 389.963,A -85,B 0,C 180,E1 -18813.263,E2 -18813.263} C_VEL
LIN {X 0,Y 247.117,Z 385.913,A -85,B 0,C 180,E1 -18815.941,E2 -18815.941} C_VEL
LIN {X 0,Y 247.284,Z 383.207,A -85,B 0,C 180,E1 -18817.35,E2 -18817.35} C_VEL
LIN {X 0,Y 247.659,Z 378.204,A -85,B 0,C 180,E1 -18819.393,E2 -18819.393} C_VEL
LIN {X 0,Y 248.232,Z 371.884,A -85,B 0,C 180,E1 -18821.433,E2 -18821.433} C_VEL
LIN {X 0,Y 248.897,Z 365.695,A -85,B 0,C 180,E1 -18823.057,E2 -18823.057} C_VEL
LIN {X 0,Y 249.676,Z 359.196,A -85,B 0,C 180,E1 -18824.469,E2 -18824.469} C_VEL
LIN {X 0,Y 250.367,Z 352.544,A -85,B 0,C 180,E1 -18825.677,E2 -18825.677} C_VEL
LIN {X 0,Y 250.164,Z 344.84,A -85,B 0,C 180,E1 -18826.871,E2 -18826.871} C_VEL
LIN {X 0,Y 249.838,Z 336.925,A -85,B 0,C 180,E1 -18827.885,E2 -18827.885} C_VEL
LIN {X 0,Y 249.264,Z 327.897,A -85,B 0,C 180,E1 -18828.815,E2 -18828.815} C_VEL
LIN {X 0,Y 248.325,Z 318.21,A -85,B 0,C 180,E1 -18829.587,E2 -18829.587} C_VEL
LIN {X 0,Y 247.64,Z 312.4,A -85,B 0,C 180,E1 -18829.973,E2 -18829.973} C_VEL
LIN {X 0,Y 248.318,Z 306.785,A -85,B 0,C 180,E1 -18834.231,E2 -18834.231} C_VEL
LIN {X 0,Y 249.309,Z 300.448,A -85,B 0,C 180,E1 -18839.083,E2 -18839.083} C_VEL
LIN {X 0,Y 250.22,Z 295.962,A -85,B 0,C 180,E1 -18842.579,E2 -18842.579} C_VEL
LIN {X 0,Y 250.402,Z 293.992,A -85,B 0,C 180,E1 -18844.15,E2 -18844.15} C_VEL
LIN {X 0,Y 249.932,Z 290.513,A -85,B 0,C 180,E1 -18847.073,E2 -18847.073} C_VEL
LIN {X 0,Y 249.148,Z 286.263,A -85,B 0,C 180,E1 -18850.986,E2 -18850.986} C_VEL
LIN {X 0,Y 249.014,Z 286.277,A -85,B 0,C 180,E1 -18855.121,E2 -18855.121} C_VEL
LIN {X 0,Y 249.018,Z 286.279,A -85,B 0,C 180,E1 -18859.521,E2 -18859.521} C_VEL
LIN {X 0,Y 249.06,Z 286.274,A -85,B 0,C 180,E1 -18863.657,E2 -18863.657} C_VEL
LIN {X 0,Y 249.049,Z 286.272,A -85,B 0,C 180,E1 -18867.845,E2 -18867.845} C_VEL
LIN {X 0,Y 249.109,Z 286.266,A -85,B 0,C 180,E1 -18871.337,E2 -18871.337} C_VEL
LIN {X 0,Y 249.146,Z 286.262,A -85,B 0,C 180,E1 -18874.965,E2 -18874.965} C_VEL
LIN {X 0,Y 249.1,Z 286.263,A -85,B 0,C 180,E1 -18878.603,E2 -18878.603} C_VEL
LIN {X 0,Y 249.187,Z 286.256,A -85,B 0,C 180,E1 -18883.616,E2 -18883.616} C_VEL
LIN {X 0,Y 249.24,Z 286.245,A -85,B 0,C 180,E1 -18888.613,E2 -18888.613} C_VEL
LIN {X 0,Y 249.451,Z 286.222,A -85,B 0,C 180,E1 -18891.899,E2 -18891.899} C_VEL
LIN {X 0,Y 249.3,Z 286.242,A -85,B 0,C 180,E1 -18895.146,E2 -18895.146} C_VEL
LIN {X 0,Y 249.682,Z 286.193,A -85,B 0,C 180,E1 -18898.384,E2 -18898.384} C_VEL
LIN {X 0,Y 249.683,Z 286.192,A -85,B 0,C 180,E1 -18901.61,E2 -18901.61} C_VEL
LIN {X 0,Y 249.457,Z 286.223,A -85,B 0,C 180,E1 -18906.728,E2 -18906.728} C_VEL
LIN {X 0,Y 249.394,Z 286.226,A -85,B 0,C 180,E1 -18909.731,E2 -18909.731} C_VEL
LIN {X 0,Y 249.206,Z 286.254,A -85,B 0,C 180,E1 -18914.7,E2 -18914.7} C_VEL
LIN {X 0,Y 249.142,Z 286.264,A -85,B 0,C 180,E1 -18918.074,E2 -18918.074} C_VEL
LIN {X 0,Y 249.089,Z 286.265,A -85,B 0,C 180,E1 -18921.514,E2 -18921.514} C_VEL
LIN {X 0,Y 249.131,Z 286.263,A -85,B 0,C 180,E1 -18925.478,E2 -18925.478} C_VEL
LIN {X 0,Y 249.079,Z 286.269,A -85,B 0,C 180,E1 -18928.988,E2 -18928.988} C_VEL
LIN {X 0,Y 249.034,Z 286.275,A -85,B 0,C 180,E1 -18932.421,E2 -18932.421} C_VEL
LIN {X 0,Y 249.073,Z 286.27,A -85,B 0,C 180,E1 -18936.334,E2 -18936.334} C_VEL
LIN {X 0,Y 249.094,Z 286.266,A -85,B 0,C 180,E1 -18940.456,E2 -18940.456} C_VEL
LIN {X 0,Y 249.089,Z 286.269,A -85,B 0,C 180,E1 -18942.81,E2 -18942.81} C_VEL
LIN {X 0,Y 249.092,Z 286.27,A -85,B 0,C 180,E1 -18947.376,E2 -18947.376} C_VEL
LIN {X 0,Y 249.045,Z 286.274,A -85,B 0,C 180,E1 -18951.621,E2 -18951.621} C_VEL
LIN {X 0,Y 249.052,Z 286.273,A -85,B 0,C 180,E1 -18955.639,E2 -18955.639} C_VEL
LIN {X 0,Y 249.042,Z 286.274,A -85,B 0,C 180,E1 -18959.47,E2 -18959.47} C_VEL
LIN {X 0,Y 249.063,Z 286.273,A -85,B 0,C 180,E1 -18963.159,E2 -18963.159} C_VEL
LIN {X 0,Y 249.064,Z 286.274,A -85,B 0,C 180,E1 -18966.729,E2 -18966.729} C_VEL
LIN {X 0,Y 248.99,Z 286.282,A -85,B 0,C 180,E1 -18970.2,E2 -18970.2} C_VEL
LIN {X 0,Y 248.767,Z 286.309,A -85,B 0,C 180,E1 -18973.837,E2 -18973.837} C_VEL
LIN {X 0,Y 248.258,Z 286.444,A -85,B 0,C 180,E1 -18977.947,E2 -18977.947} C_VEL
LIN {X 0,Y 248.224,Z 290.036,A -85,B 0,C 180,E1 -18982.26,E2 -18982.26} C_VEL
LIN {X 0,Y 248.012,Z 291.711,A -85,B 0,C 180,E1 -18984.204,E2 -18984.204} C_VEL
LIN {X 0,Y 250.095,Z 302.557,A -85,B 0,C 180,E1 -18985.061,E2 -18985.061} C_VEL
LIN {X 0,Y 251.372,Z 311.726,A -85,B 0,C 180,E1 -18985.99,E2 -18985.99} C_VEL
LIN {X 0,Y 252.238,Z 319.845,A -85,B 0,C 180,E1 -18987.003,E2 -18987.003} C_VEL
LIN {X 0,Y 251.415,Z 328.19,A -85,B 0,C 180,E1 -18988.196,E2 -18988.196} C_VEL
LIN {X 0,Y 250.522,Z 336.097,A -85,B 0,C 180,E1 -18989.596,E2 -18989.596} C_VEL
LIN {X 0,Y 249.64,Z 343.481,A -85,B 0,C 180,E1 -18991.208,E2 -18991.208} C_VEL
LIN {X 0,Y 248.755,Z 350.961,A -85,B 0,C 180,E1 -18993.237,E2 -18993.237} C_VEL
LIN {X 0,Y 248.162,Z 356.807,A -85,B 0,C 180,E1 -18995.279,E2 -18995.279} C_VEL
LIN {X 0,Y 247.624,Z 361.446,A -85,B 0,C 180,E1 -18997.34,E2 -18997.34} C_VEL
LIN {X 0,Y 247.283,Z 364.446,A -85,B 0,C 180,E1 -18998.991,E2 -18998.991} C_VEL
LIN {X 0,Y 246.93,Z 367.702,A -85,B 0,C 180,E1 -19001.49,E2 -19001.49} C_VEL
LIN {X 0,Y 246.902,Z 369.241,A -85,B 0,C 180,E1 -19003.16,E2 -19003.16} C_VEL
LIN {X 0,Y 246.969,Z 370.238,A -85,B 0,C 180,E1 -19004.837,E2 -19004.837} C_VEL
LIN {X 0,Y 247.082,Z 370.639,A -85,B 0,C 180,E1 -19006.523,E2 -19006.523} C_VEL
LIN {X 0,Y 247.351,Z 370.532,A -85,B 0,C 180,E1 -19008.21,E2 -19008.21} C_VEL
LIN {X 0,Y 248.121,Z 369.393,A -85,B 0,C 180,E1 -19010.828,E2 -19010.828} C_VEL
LIN {X 0,Y 249.07,Z 367.138,A -85,B 0,C 180,E1 -19013.266,E2 -19013.266} C_VEL
LIN {X 0,Y 250.273,Z 363.761,A -85,B 0,C 180,E1 -19015.576,E2 -19015.576} C_VEL
LIN {X 0,Y 251.514,Z 360.092,A -85,B 0,C 180,E1 -19017.453,E2 -19017.453} C_VEL
LIN {X 0,Y 253.145,Z 354.842,A -85,B 0,C 180,E1 -19019.521,E2 -19019.521} C_VEL
LIN {X 0,Y 254.516,Z 349.779,A -85,B 0,C 180,E1 -19021.136,E2 -19021.136} C_VEL
LIN {X 0,Y 256.323,Z 343.333,A -85,B 0,C 180,E1 -19022.784,E2 -19022.784} C_VEL
LIN {X 0,Y 257.933,Z 336.637,A -85,B 0,C 180,E1 -19024.19,E2 -19024.19} C_VEL
LIN {X 0,Y 258.908,Z 332.533,A -85,B 0,C 180,E1 -19024.941,E2 -19024.941} C_VEL
LIN {X 0,Y 257.92,Z 324.22,A -85,B 0,C 180,E1 -19026.509,E2 -19026.509} C_VEL
LIN {X 0,Y 256.296,Z 316.225,A -85,B 0,C 180,E1 -19027.862,E2 -19027.862} C_VEL
LIN {X 0,Y 253.893,Z 307.366,A -85,B 0,C 180,E1 -19029.195,E2 -19029.195} C_VEL
LIN {X 0,Y 250.728,Z 298.447,A -85,B 0,C 180,E1 -19030.418,E2 -19030.418} C_VEL
LIN {X 0,Y 248.84,Z 293.124,A -85,B 0,C 180,E1 -19031.069,E2 -19031.069} C_VEL
LIN {X 0,Y 248.952,Z 291.664,A -85,B 0,C 180,E1 -19032.784,E2 -19032.784} C_VEL
LIN {X 0,Y 249.129,Z 289.992,A -85,B 0,C 180,E1 -19035.155,E2 -19035.155} C_VEL
LIN {X 0,Y 249.146,Z 288.495,A -85,B 0,C 180,E1 -19037.395,E2 -19037.395} C_VEL
LIN {X 0,Y 249.052,Z 287.079,A -85,B 0,C 180,E1 -19039.629,E2 -19039.629} C_VEL
LIN {X 0,Y 249.033,Z 286.281,A -85,B 0,C 180,E1 -19042.199,E2 -19042.199} C_VEL
LIN {X 0,Y 249.044,Z 286.277,A -85,B 0,C 180,E1 -19045.644,E2 -19045.644} C_VEL
LIN {X 0,Y 249.03,Z 286.277,A -85,B 0,C 180,E1 -19049.474,E2 -19049.474} C_VEL
LIN {X 0,Y 249.052,Z 286.274,A -85,B 0,C 180,E1 -19053.164,E2 -19053.164} C_VEL
LIN {X 0,Y 249.046,Z 286.273,A -85,B 0,C 180,E1 -19056.733,E2 -19056.733} C_VEL
LIN {X 0,Y 249.094,Z 286.269,A -85,B 0,C 180,E1 -19060.214,E2 -19060.214} C_VEL
LIN {X 0,Y 249.228,Z 286.254,A -85,B 0,C 180,E1 -19063.624,E2 -19063.624} C_VEL
LIN {X 0,Y 249.232,Z 286.25,A -85,B 0,C 180,E1 -19068.619,E2 -19068.619} C_VEL
LIN {X 0,Y 249.426,Z 286.228,A -85,B 0,C 180,E1 -19071.904,E2 -19071.904} C_VEL
LIN {X 0,Y 249.279,Z 286.246,A -85,B 0,C 180,E1 -19075.151,E2 -19075.151} C_VEL
LIN {X 0,Y 249.666,Z 286.192,A -85,B 0,C 180,E1 -19078.39,E2 -19078.39} C_VEL
LIN {X 0,Y 249.666,Z 286.192,A -85,B 0,C 180,E1 -19081.616,E2 -19081.616} C_VEL
LIN {X 0,Y 249.453,Z 286.218,A -85,B 0,C 180,E1 -19086.473,E2 -19086.473} C_VEL
LIN {X 0,Y 249.416,Z 286.229,A -85,B 0,C 180,E1 -19089.736,E2 -19089.736} C_VEL
LIN {X 0,Y 249.199,Z 286.257,A -85,B 0,C 180,E1 -19094.706,E2 -19094.706} C_VEL
LIN {X 0,Y 249.133,Z 286.266,A -85,B 0,C 180,E1 -19098.08,E2 -19098.08} C_VEL
LIN {X 0,Y 249.078,Z 286.273,A -85,B 0,C 180,E1 -19101.522,E2 -19101.522} C_VEL
LIN {X 0,Y 249.08,Z 286.274,A -85,B 0,C 180,E1 -19105.463,E2 -19105.463} C_VEL
LIN {X 0,Y 249.032,Z 286.283,A -85,B 0,C 180,E1 -19108.977,E2 -19108.977} C_VEL
LIN {X 0,Y 249.008,Z 286.283,A -85,B 0,C 180,E1 -19113.021,E2 -19113.021} C_VEL
LIN {X 0,Y 249.071,Z 286.277,A -85,B 0,C 180,E1 -19116.341,E2 -19116.341} C_VEL
LIN {X 0,Y 249.114,Z 286.453,A -85,B 0,C 180,E1 -19118.367,E2 -19118.367} C_VEL
LIN {X 0,Y 249.291,Z 287.707,A -85,B 0,C 180,E1 -19120.003,E2 -19120.003} C_VEL
LIN {X 0,Y 248.848,Z 288.908,A -85,B 0,C 180,E1 -19121.327,E2 -19121.327} C_VEL
LIN {X 0,Y 246.327,Z 291.301,A -85,B 0,C 180,E1 -19123.473,E2 -19123.473} C_VEL
LIN {X 0,Y 244.149,Z 293.298,A -85,B 0,C 180,E1 -19125.216,E2 -19125.216} C_VEL
LIN {X 0,Y 243.296,Z 294.695,A -85,B 0,C 180,E1 -19126.567,E2 -19126.567} C_VEL
LIN {X 0,Y 243.276,Z 295.122,A -85,B 0,C 180,E1 -19127.025,E2 -19127.025} C_VEL
LIN {X 0,Y 244.025,Z 298.862,A -85,B 0,C 180,E1 -19131.046,E2 -19131.046} C_VEL
LIN {X 0,Y 244.414,Z 301.469,A -85,B 0,C 180,E1 -19133.626,E2 -19133.626} C_VEL
LIN {X 0,Y 244.547,Z 302.822,A -85,B 0,C 180,E1 -19134.919,E2 -19134.919} C_VEL
LIN {X 0,Y 244.341,Z 304.971,A -85,B 0,C 180,E1 -19136.876,E2 -19136.876} C_VEL
LIN {X 0,Y 242.918,Z 310.364,A -85,B 0,C 180,E1 -19141.489,E2 -19141.489} C_VEL
LIN {X 0,Y 242.769,Z 311.011,A -85,B 0,C 180,E1 -19142.029,E2 -19142.029} C_VEL
LIN {X 0,Y 243.609,Z 314.325,A -85,B 0,C 180,E1 -19142.353,E2 -19142.353} C_VEL
LIN {X 0,Y 246.029,Z 324.02,A -85,B 0,C 180,E1 -19143.47,E2 -19143.47} C_VEL
LIN {X 0,Y 247.755,Z 333.218,A -85,B 0,C 180,E1 -19144.68,E2 -19144.68} C_VEL
LIN {X 0,Y 248.855,Z 342.236,A -85,B 0,C 180,E1 -19146.035,E2 -19146.035} C_VEL
LIN {X 0,Y 249.258,Z 350.266,A -85,B 0,C 180,E1 -19147.411,E2 -19147.411} C_VEL
LIN {X 0,Y 249.189,Z 356.196,A -85,B 0,C 180,E1 -19148.551,E2 -19148.551} C_VEL
LIN {X 0,Y 248.657,Z 362.208,A -85,B 0,C 180,E1 -19149.838,E2 -19149.838} C_VEL
LIN {X 0,Y 246.567,Z 369.881,A -85,B 0,C 180,E1 -19151.73,E2 -19151.73} C_VEL
LIN {X 0,Y 244.953,Z 375.169,A -85,B 0,C 180,E1 -19153.329,E2 -19153.329} C_VEL
LIN {X 0,Y 243.586,Z 379.597,A -85,B 0,C 180,E1 -19154.952,E2 -19154.952} C_VEL
LIN {X 0,Y 242.003,Z 384.832,A -85,B 0,C 180,E1 -19157.422,E2 -19157.422} C_VEL
LIN {X 0,Y 241.196,Z 387.546,A -85,B 0,C 180,E1 -19159.085,E2 -19159.085} C_VEL
LIN {X 0,Y 240.35,Z 390.546,A -85,B 0,C 180,E1 -19161.595,E2 -19161.595} C_VEL
LIN {X 0,Y 240.039,Z 391.895,A -85,B 0,C 180,E1 -19163.277,E2 -19163.277} C_VEL
LIN {X 0,Y 239.887,Z 392.782,A -85,B 0,C 180,E1 -19164.96,E2 -19164.96} C_VEL
LIN {X 0,Y 239.904,Z 393.146,A -85,B 0,C 180,E1 -19166.643,E2 -19166.643} C_VEL
LIN {X 0,Y 239.982,Z 392.943,A -85,B 0,C 180,E1 -19168.324,E2 -19168.324} C_VEL
LIN {X 0,Y 240.025,Z 392.274,A -85,B 0,C 180,E1 -19170.002,E2 -19170.002} C_VEL
LIN {X 0,Y 240.022,Z 391.124,A -85,B 0,C 180,E1 -19171.68,E2 -19171.68} C_VEL
LIN {X 0,Y 240.016,Z 389.458,A -85,B 0,C 180,E1 -19173.359,E2 -19173.359} C_VEL
LIN {X 0,Y 240.033,Z 385.892,A -85,B 0,C 180,E1 -19175.8,E2 -19175.8} C_VEL
LIN {X 0,Y 240.212,Z 382.545,A -85,B 0,C 180,E1 -19177.568,E2 -19177.568} C_VEL
LIN {X 0,Y 240.626,Z 377.459,A -85,B 0,C 180,E1 -19179.67,E2 -19179.67} C_VEL
LIN {X 0,Y 241.107,Z 372.487,A -85,B 0,C 180,E1 -19181.349,E2 -19181.349} C_VEL
LIN {X 0,Y 241.747,Z 366.482,A -85,B 0,C 180,E1 -19183.023,E2 -19183.023} C_VEL
LIN {X 0,Y 242.649,Z 359.176,A -85,B 0,C 180,E1 -19184.683,E2 -19184.683} C_VEL
LIN {X 0,Y 243.326,Z 352.58,A -85,B 0,C 180,E1 -19185.928,E2 -19185.928} C_VEL
LIN {X 0,Y 243.156,Z 345.138,A -85,B 0,C 180,E1 -19187.13,E2 -19187.13} C_VEL
LIN {X 0,Y 242.818,Z 337.049,A -85,B 0,C 180,E1 -19188.213,E2 -19188.213} C_VEL
LIN {X 0,Y 242.295,Z 328.284,A -85,B 0,C 180,E1 -19189.157,E2 -19189.157} C_VEL
LIN {X 0,Y 241.383,Z 318.545,A -85,B 0,C 180,E1 -19189.973,E2 -19189.973} C_VEL
LIN {X 0,Y 240.634,Z 312.13,A -85,B 0,C 180,E1 -19190.407,E2 -19190.407} C_VEL
LIN {X 0,Y 241.476,Z 305.562,A -85,B 0,C 180,E1 -19195.542,E2 -19195.542} C_VEL
LIN {X 0,Y 242.56,Z 299.322,A -85,B 0,C 180,E1 -19200.47,E2 -19200.47} C_VEL
LIN {X 0,Y 243.216,Z 295.861,A -85,B 0,C 180,E1 -19203.302,E2 -19203.302} C_VEL
LIN {X 0,Y 243.212,Z 293.463,A -85,B 0,C 180,E1 -19205.307,E2 -19205.307} C_VEL
LIN {X 0,Y 242.594,Z 289.855,A -85,B 0,C 180,E1 -19208.535,E2 -19208.535} C_VEL
LIN {X 0,Y 242.118,Z 287.138,A -85,B 0,C 180,E1 -19211.114,E2 -19211.114} C_VEL
LIN {X 0,Y 241.946,Z 287.157,A -85,B 0,C 180,E1 -19216.571,E2 -19216.571} C_VEL
LIN {X 0,Y 241.968,Z 287.155,A -85,B 0,C 180,E1 -19220.28,E2 -19220.28} C_VEL
LIN {X 0,Y 241.999,Z 287.151,A -85,B 0,C 180,E1 -19224.488,E2 -19224.488} C_VEL
LIN {X 0,Y 241.986,Z 287.15,A -85,B 0,C 180,E1 -19228.479,E2 -19228.479} C_VEL
LIN {X 0,Y 242.019,Z 287.148,A -85,B 0,C 180,E1 -19232.311,E2 -19232.311} C_VEL
LIN {X 0,Y 242.052,Z 287.142,A -85,B 0,C 180,E1 -19236.013,E2 -19236.013} C_VEL
LIN {X 0,Y 242.027,Z 287.147,A -85,B 0,C 180,E1 -19239.604,E2 -19239.604} C_VEL
LIN {X 0,Y 242.126,Z 287.138,A -85,B 0,C 180,E1 -19243.314,E2 -19243.314} C_VEL
LIN {X 0,Y 242.174,Z 287.124,A -85,B 0,C 180,E1 -19248.276,E2 -19248.276} C_VEL
LIN {X 0,Y 242.399,Z 287.101,A -85,B 0,C 180,E1 -19251.662,E2 -19251.662} C_VEL
LIN {X 0,Y 242.26,Z 287.12,A -85,B 0,C 180,E1 -19255.004,E2 -19255.004} C_VEL
LIN {X 0,Y 242.643,Z 287.069,A -85,B 0,C 180,E1 -19258.337,E2 -19258.337} C_VEL
LIN {X 0,Y 242.644,Z 287.069,A -85,B 0,C 180,E1 -19261.657,E2 -19261.657} C_VEL
LIN {X 0,Y 242.437,Z 287.097,A -85,B 0,C 180,E1 -19266.704,E2 -19266.704} C_VEL
LIN {X 0,Y 242.32,Z 287.109,A -85,B 0,C 180,E1 -19270.018,E2 -19270.018} C_VEL
LIN {X 0,Y 242.168,Z 287.13,A -85,B 0,C 180,E1 -19275.137,E2 -19275.137} C_VEL
LIN {X 0,Y 242.076,Z 287.141,A -85,B 0,C 180,E1 -19278.62,E2 -19278.62} C_VEL
LIN {X 0,Y 242.015,Z 287.147,A -85,B 0,C 180,E1 -19282.176,E2 -19282.176} C_VEL
LIN {X 0,Y 242.067,Z 287.146,A -85,B 0,C 180,E1 -19285.834,E2 -19285.834} C_VEL
LIN {X 0,Y 242.028,Z 287.15,A -85,B 0,C 180,E1 -19289.576,E2 -19289.576} C_VEL
LIN {X 0,Y 241.989,Z 287.156,A -85,B 0,C 180,E1 -19293.487,E2 -19293.487} C_VEL
LIN {X 0,Y 242.017,Z 287.152,A -85,B 0,C 180,E1 -19297.572,E2 -19297.572} C_VEL
LIN {X 0,Y 242.036,Z 287.147,A -85,B 0,C 180,E1 -19301.896,E2 -19301.896} C_VEL
LIN {X 0,Y 242.018,Z 287.148,A -85,B 0,C 180,E1 -19306.545,E2 -19306.545} C_VEL
LIN {X 0,Y 242.003,Z 287.149,A -85,B 0,C 180,E1 -19310.288,E2 -19310.288} C_VEL
LIN {X 0,Y 242.028,Z 287.147,A -85,B 0,C 180,E1 -19314.494,E2 -19314.494} C_VEL
LIN {X 0,Y 241.966,Z 287.156,A -85,B 0,C 180,E1 -19318.476,E2 -19318.476} C_VEL
LIN {X 0,Y 241.998,Z 287.152,A -85,B 0,C 180,E1 -19322.309,E2 -19322.309} C_VEL
LIN {X 0,Y 242.044,Z 287.146,A -85,B 0,C 180,E1 -19326.012,E2 -19326.012} C_VEL
LIN {X 0,Y 241.959,Z 287.156,A -85,B 0,C 180,E1 -19329.599,E2 -19329.599} C_VEL
LIN {X 0,Y 241.73,Z 287.185,A -85,B 0,C 180,E1 -19333.61,E2 -19333.61} C_VEL
LIN {X 0,Y 241.219,Z 287.304,A -85,B 0,C 180,E1 -19338.017,E2 -19338.017} C_VEL
LIN {X 0,Y 241.168,Z 290.719,A -85,B 0,C 180,E1 -19342.196,E2 -19342.196} C_VEL
LIN {X 0,Y 241.014,Z 292.081,A -85,B 0,C 180,E1 -19343.773,E2 -19343.773} C_VEL
LIN {X 0,Y 243.212,Z 303.538,A -85,B 0,C 180,E1 -19344.713,E2 -19344.713} C_VEL
LIN {X 0,Y 244.457,Z 312.563,A -85,B 0,C 180,E1 -19345.67,E2 -19345.67} C_VEL
LIN {X 0,Y 245.272,Z 320.589,A -85,B 0,C 180,E1 -19346.713,E2 -19346.713} C_VEL
LIN {X 0,Y 244.446,Z 328.853,A -85,B 0,C 180,E1 -19347.938,E2 -19347.938} C_VEL
LIN {X 0,Y 243.601,Z 335.687,A -85,B 0,C 180,E1 -19349.171,E2 -19349.171} C_VEL
LIN {X 0,Y 242.936,Z 341.47,A -85,B 0,C 180,E1 -19350.412,E2 -19350.412} C_VEL
LIN {X 0,Y 242.157,Z 347.917,A -85,B 0,C 180,E1 -19352.077,E2 -19352.077} C_VEL
LIN {X 0,Y 241.476,Z 353.285,A -85,B 0,C 180,E1 -19353.752,E2 -19353.752} C_VEL
LIN {X 0,Y 240.902,Z 358.724,A -85,B 0,C 180,E1 -19355.858,E2 -19355.858} C_VEL
LIN {X 0,Y 240.475,Z 362.26,A -85,B 0,C 180,E1 -19357.554,E2 -19357.554} C_VEL
LIN {X 0,Y 240.006,Z 366.337,A -85,B 0,C 180,E1 -19360.117,E2 -19360.117} C_VEL
LIN {X 0,Y 239.825,Z 368.3,A -85,B 0,C 180,E1 -19361.835,E2 -19361.835} C_VEL
LIN {X 0,Y 239.871,Z 370.467,A -85,B 0,C 180,E1 -19364.806,E2 -19364.806} C_VEL
LIN {X 0,Y 240.055,Z 371.03,A -85,B 0,C 180,E1 -19367.021,E2 -19367.021} C_VEL
LIN {X 0,Y 240.382,Z 370.818,A -85,B 0,C 180,E1 -19368.758,E2 -19368.758} C_VEL
LIN {X 0,Y 241.122,Z 369.74,A -85,B 0,C 180,E1 -19371.151,E2 -19371.151} C_VEL
LIN {X 0,Y 242.292,Z 367.114,A -85,B 0,C 180,E1 -19373.957,E2 -19373.957} C_VEL
LIN {X 0,Y 243.226,Z 364.736,A -85,B 0,C 180,E1 -19375.682,E2 -19375.682} C_VEL
LIN {X 0,Y 244.948,Z 359.795,A -85,B 0,C 180,E1 -19378.254,E2 -19378.254} C_VEL
LIN {X 0,Y 246.337,Z 355.609,A -85,B 0,C 180,E1 -19379.949,E2 -19379.949} C_VEL
LIN {X 0,Y 247.933,Z 350.115,A -85,B 0,C 180,E1 -19381.753,E2 -19381.753} C_VEL
LIN {X 0,Y 249.658,Z 344.307,A -85,B 0,C 180,E1 -19383.291,E2 -19383.291} C_VEL
LIN {X 0,Y 251.599,Z 336.69,A -85,B 0,C 180,E1 -19384.931,E2 -19384.931} C_VEL
LIN {X 0,Y 252.286,Z 333.503,A -85,B 0,C 180,E1 -19385.55,E2 -19385.55} C_VEL
LIN {X 0,Y 251.07,Z 324.001,A -85,B 0,C 180,E1 -19387.421,E2 -19387.421} C_VEL
LIN {X 0,Y 249.294,Z 315.565,A -85,B 0,C 180,E1 -19388.888,E2 -19388.888} C_VEL
LIN {X 0,Y 247.061,Z 307.554,A -85,B 0,C 180,E1 -19390.144,E2 -19390.144} C_VEL
LIN {X 0,Y 243.63,Z 298.251,A -85,B 0,C 180,E1 -19391.493,E2 -19391.493} C_VEL
LIN {X 0,Y 241.897,Z 293.231,A -85,B 0,C 180,E1 -19392.155,E2 -19392.155} C_VEL
LIN {X 0,Y 242.133,Z 290.275,A -85,B 0,C 180,E1 -19396.518,E2 -19396.518} C_VEL
LIN {X 0,Y 242.016,Z 287.927,A -85,B 0,C 180,E1 -19400.298,E2 -19400.298} C_VEL
LIN {X 0,Y 241.98,Z 287.16,A -85,B 0,C 180,E1 -19401.641,E2 -19401.641} C_VEL
LIN {X 0,Y 242.019,Z 287.153,A -85,B 0,C 180,E1 -19404.499,E2 -19404.499} C_VEL
LIN {X 0,Y 241.958,Z 287.16,A -85,B 0,C 180,E1 -19408.482,E2 -19408.482} C_VEL
LIN {X 0,Y 241.985,Z 287.157,A -85,B 0,C 180,E1 -19412.314,E2 -19412.314} C_VEL
LIN {X 0,Y 242.025,Z 287.146,A -85,B 0,C 180,E1 -19416.016,E2 -19416.016} C_VEL
LIN {X 0,Y 242.021,Z 287.147,A -85,B 0,C 180,E1 -19419.61,E2 -19419.61} C_VEL
LIN {X 0,Y 242.149,Z 287.132,A -85,B 0,C 180,E1 -19423.281,E2 -19423.281} C_VEL
LIN {X 0,Y 242.168,Z 287.131,A -85,B 0,C 180,E1 -19428.282,E2 -19428.282} C_VEL
LIN {X 0,Y 242.375,Z 287.107,A -85,B 0,C 180,E1 -19431.667,E2 -19431.667} C_VEL
LIN {X 0,Y 242.239,Z 287.123,A -85,B 0,C 180,E1 -19435.01,E2 -19435.01} C_VEL
LIN {X 0,Y 242.626,Z 287.068,A -85,B 0,C 180,E1 -19438.343,E2 -19438.343} C_VEL
LIN {X 0,Y 242.626,Z 287.069,A -85,B 0,C 180,E1 -19441.663,E2 -19441.663} C_VEL
LIN {X 0,Y 242.425,Z 287.094,A -85,B 0,C 180,E1 -19446.662,E2 -19446.662} C_VEL
LIN {X 0,Y 242.338,Z 287.112,A -85,B 0,C 180,E1 -19450.024,E2 -19450.024} C_VEL
LIN {X 0,Y 242.16,Z 287.133,A -85,B 0,C 180,E1 -19455.144,E2 -19455.144} C_VEL
LIN {X 0,Y 242.066,Z 287.144,A -85,B 0,C 180,E1 -19458.627,E2 -19458.627} C_VEL
LIN {X 0,Y 241.999,Z 287.153,A -85,B 0,C 180,E1 -19462.184,E2 -19462.184} C_VEL
LIN {X 0,Y 242.027,Z 287.154,A -85,B 0,C 180,E1 -19465.824,E2 -19465.824} C_VEL
LIN {X 0,Y 241.964,Z 287.164,A -85,B 0,C 180,E1 -19469.592,E2 -19469.592} C_VEL
LIN {X 0,Y 241.986,Z 287.163,A -85,B 0,C 180,E1 -19473.494,E2 -19473.494} C_VEL
LIN {X 0,Y 242.037,Z 287.259,A -85,B 0,C 180,E1 -19477.314,E2 -19477.314} C_VEL
LIN {X 0,Y 242.567,Z 290.647,A -85,B 0,C 180,E1 -19481.792,E2 -19481.792} C_VEL
LIN {X 0,Y 243.195,Z 294.433,A -85,B 0,C 180,E1 -19486.261,E2 -19486.261} C_VEL
LIN {X 0,Y 243.276,Z 295.122,A -85,B 0,C 180,E1 -19487.025,E2 -19487.025} C_VEL
LIN {X 0,Y 242.83,Z 296.476,A -85,B 0,C 180,E1 -19488.376,E2 -19488.376} C_VEL
LIN {X 0,Y 240.409,Z 299.048,A -85,B 0,C 180,E1 -19490.573,E2 -19490.573} C_VEL
LIN {X 0,Y 237.651,Z 302.226,A -85,B 0,C 180,E1 -19493.27,E2 -19493.27} C_VEL
LIN {X 0,Y 237.449,Z 303.212,A -85,B 0,C 180,E1 -19494.2,E2 -19494.2} C_VEL
LIN {X 0,Y 237.425,Z 305.074,A -85,B 0,C 180,E1 -19495.982,E2 -19495.982} C_VEL
LIN {X 0,Y 236.405,Z 309.183,A -85,B 0,C 180,E1 -19499.646,E2 -19499.646} C_VEL
